C07319=1124.447,364.307,-84.895,-177.079,11.092,149.484
C07320=1124.444,364.554,-84.931,-177.076,11.094,149.483
C07321=1124.440,364.802,-84.967,-177.072,11.097,149.483
C07322=1124.436,365.049,-85.004,-177.069,11.099,149.483
C07323=1124.432,365.296,-85.040,-177.065,11.101,149.483
C07324=1124.429,365.543,-85.076,-177.062,11.104,149.482
C07325=1124.425,365.791,-85.113,-177.059,11.106,149.482
C07326=1124.421,366.038,-85.148,-177.056,11.109,149.482
C07327=1124.417,366.285,-85.185,-177.052,11.111,149.482
C07328=1124.413,366.532,-85.221,-177.050,11.113,149.482
C07329=1124.409,366.779,-85.258,-177.046,11.115,149.481
C07330=1124.406,367.027,-85.294,-177.043,11.118,149.481
C07331=1124.402,367.274,-85.331,-177.039,11.120,149.481
C07332=1124.398,367.522,-85.368,-177.036,11.123,149.480
C07333=1124.394,367.769,-85.403,-177.033,11.125,149.480
C07334=1124.390,368.017,-85.440,-177.029,11.128,149.480
C07335=1124.387,368.264,-85.477,-177.026,11.130,149.480
C07336=1124.383,368.511,-85.513,-177.023,11.132,149.480
C07337=1124.379,368.758,-85.550,-177.020,11.134,149.479
C07338=1124.375,369.005,-85.586,-177.017,11.137,149.479
C07339=1124.372,369.253,-85.623,-177.014,11.139,149.479
C07340=1124.368,369.500,-85.659,-177.010,11.142,149.479
C07341=1124.364,369.747,-85.696,-177.007,11.144,149.479
C07342=1124.360,369.995,-85.733,-177.004,11.146,149.478
C07343=1124.357,370.241,-85.769,-177.001,11.148,149.478
C07344=1124.353,370.489,-85.806,-176.998,11.151,149.478
C07345=1124.349,370.737,-85.843,-176.994,11.153,149.478
C07346=1124.346,370.983,-85.880,-176.991,11.156,149.477
C07347=1124.342,371.231,-85.917,-176.988,11.158,149.477
C07348=1124.338,371.478,-85.953,-176.985,11.160,149.477
C07349=1124.333,371.725,-85.990,-176.982,11.162,149.477
C07350=1124.331,371.973,-86.027,-176.978,11.165,149.477
C07351=1124.327,372.220,-86.064,-176.975,11.167,149.476
C07352=1124.323,372.467,-86.101,-176.972,11.170,149.476
C07353=1124.318,372.714,-86.137,-176.969,11.171,149.476
C07354=1124.315,372.961,-86.174,-176.966,11.174,149.476
C07355=1124.312,373.209,-86.211,-176.963,11.176,149.476
C07356=1124.308,373.456,-86.248,-176.960,11.179,149.476
C07357=1124.303,373.703,-86.285,-176.956,11.182,149.475
C07358=1124.300,373.950,-86.321,-176.954,11.183,149.475
C07359=1124.297,374.198,-86.358,-176.950,11.186,149.475
C07360=1124.292,374.445,-86.395,-176.947,11.188,149.475
C07361=1124.288,374.692,-86.432,-176.944,11.191,149.474
C07362=1124.285,374.939,-86.469,-176.942,11.193,149.474
C07363=1124.282,375.152,-86.501,-176.938,11.195,149.474
C07364=1124.279,375.364,-86.533,-176.936,11.197,149.474
C07365=1124.275,375.577,-86.565,-176.933,11.199,149.474
C07366=1124.272,375.789,-86.597,-176.931,11.201,149.474
C07367=1124.269,376.001,-86.628,-176.928,11.204,149.474
C07368=1124.266,376.214,-86.660,-176.925,11.205,149.473
C07369=1124.262,376.426,-86.691,-176.923,11.207,149.473
C07370=1124.259,376.638,-86.723,-176.921,11.209,149.473
C07371=1124.256,376.886,-86.761,-176.917,11.212,149.473
C07372=1124.252,377.132,-86.798,-176.914,11.214,149.473
C07373=1124.248,377.379,-86.835,-176.911,11.216,149.473
C07374=1124.244,377.626,-86.872,-176.908,11.219,149.473
C07375=1124.241,377.874,-86.910,-176.905,11.221,149.472
C07376=1124.237,378.121,-86.947,-176.902,11.224,149.472
C07377=1124.233,378.368,-86.984,-176.900,11.226,149.472
C07378=1124.229,378.615,-87.021,-176.896,11.228,149.472
C07379=1124.225,378.863,-87.058,-176.893,11.231,149.472
C07380=1124.221,379.110,-87.095,-176.890,11.234,149.472
C07381=1124.218,379.357,-87.133,-176.888,11.236,149.472
C07382=1124.214,379.604,-87.170,-176.884,11.238,149.471
C07383=1124.211,379.852,-87.208,-176.882,11.241,149.471
C07384=1124.207,380.099,-87.245,-176.878,11.243,149.471
C07385=1124.203,380.345,-87.282,-176.876,11.245,149.471
C07386=1124.199,380.593,-87.320,-176.873,11.248,149.471
C07387=1124.196,380.840,-87.357,-176.870,11.251,149.471
C07388=1124.191,381.087,-87.394,-176.867,11.252,149.471
C07389=1124.188,381.334,-87.432,-176.864,11.255,149.471
C07390=1124.184,381.581,-87.469,-176.861,11.258,149.471
C07391=1124.181,381.829,-87.507,-176.858,11.261,149.471
C07392=1124.177,382.076,-87.544,-176.856,11.263,149.471
C07393=1124.174,382.323,-87.582,-176.853,11.265,149.470
C07394=1124.170,382.570,-87.618,-176.850,11.268,149.470
C07395=1124.166,382.817,-87.656,-176.847,11.270,149.470
C07396=1124.163,383.064,-87.694,-176.844,11.273,149.470
C07397=1124.158,383.312,-87.731,-176.841,11.275,149.470
C07398=1124.155,383.559,-87.769,-176.839,11.278,149.470
C07399=1124.151,383.806,-87.807,-176.837,11.280,149.470
C07400=1124.147,384.053,-87.844,-176.836,11.281,149.470
C07401=1124.144,384.300,-87.882,-176.833,11.283,149.470
C07402=1124.140,384.547,-87.919,-176.832,11.285,149.470
C07403=1124.136,384.794,-87.956,-176.830,11.287,149.470
C07404=1124.132,385.041,-87.994,-176.828,11.289,149.471
C07405=1124.129,385.289,-88.033,-176.827,11.291,149.470
C07406=1124.124,385.536,-88.069,-176.825,11.293,149.471
C07407=1124.121,385.783,-88.107,-176.823,11.295,149.471
C07408=1124.117,386.030,-88.145,-176.822,11.297,149.471
C07409=1124.114,386.277,-88.183,-176.820,11.299,149.471
C07410=1124.110,386.524,-88.220,-176.818,11.302,149.471
C07411=1124.106,386.772,-88.258,-176.816,11.304,149.471
C07412=1124.102,387.018,-88.296,-176.815,11.306,149.471
C07413=1124.099,387.265,-88.334,-176.813,11.308,149.471
C07414=1124.095,387.513,-88.371,-176.812,11.311,149.472
C07415=1124.092,387.760,-88.409,-176.810,11.312,149.472
C07416=1124.088,388.007,-88.446,-176.808,11.315,149.472
C07417=1124.084,388.254,-88.485,-176.807,11.317,149.472
C07418=1124.080,388.501,-88.522,-176.805,11.320,149.472
C07419=1124.077,388.713,-88.555,-176.804,11.321,149.472
C07420=1124.074,388.925,-88.587,-176.803,11.323,149.473
C07421=1124.071,389.137,-88.619,-176.801,11.325,149.473
C07422=1124.068,389.349,-88.651,-176.800,11.327,149.473
C07423=1124.065,389.562,-88.684,-176.798,11.330,149.473
C07424=1124.061,389.774,-88.717,-176.797,11.331,149.473
C07425=1124.059,389.987,-88.749,-176.796,11.333,149.474
C07426=1124.054,390.323,-88.801,-176.794,11.337,149.474
C07427=1124.050,390.571,-88.838,-176.792,11.339,149.474
C07428=1124.046,390.817,-88.877,-176.791,11.342,149.474
C07429=1124.042,391.065,-88.915,-176.789,11.344,149.475
C07430=1124.039,391.311,-88.952,-176.788,11.346,149.475
C07431=1124.035,391.559,-88.990,-176.787,11.349,149.475
C07432=1124.031,391.805,-89.028,-176.786,11.352,149.476
C07433=1124.028,392.053,-89.066,-176.784,11.354,149.476
C07434=1124.025,392.300,-89.104,-176.783,11.357,149.476
C07435=1124.020,392.547,-89.142,-176.781,11.360,149.477
C07436=1124.017,392.794,-89.180,-176.780,11.362,149.477
C07437=1124.013,393.041,-89.218,-176.778,11.365,149.477
C07438=1124.010,393.288,-89.256,-176.778,11.367,149.478
C07439=1124.005,393.535,-89.294,-176.776,11.370,149.478
C07440=1124.002,393.782,-89.332,-176.775,11.373,149.478
C07441=1123.998,394.030,-89.370,-176.774,11.376,149.479
C07442=1123.994,394.276,-89.408,-176.772,11.378,149.479
C07443=1123.991,394.524,-89.446,-176.771,11.381,149.480
C07444=1123.987,394.770,-89.484,-176.770,11.384,149.480
C07445=1123.984,395.018,-89.522,-176.768,11.387,149.481
C07446=1123.980,395.265,-89.560,-176.767,11.390,149.481
C07447=1123.976,395.512,-89.598,-176.766,11.393,149.481
C07448=1123.973,395.759,-89.636,-176.765,11.396,149.482
C07449=1123.969,396.005,-89.674,-176.763,11.399,149.482
C07450=1123.965,396.253,-89.713,-176.762,11.402,149.483
C07451=1123.962,396.500,-89.751,-176.761,11.405,149.483
C07452=1123.958,396.747,-89.789,-176.760,11.408,149.484
C07453=1123.954,396.994,-89.827,-176.759,11.411,149.484
C07454=1123.951,397.241,-89.864,-176.758,11.414,149.485
C07455=1123.947,397.488,-89.903,-176.757,11.417,149.485
C07456=1123.943,397.735,-89.941,-176.756,11.420,149.486
C07457=1123.939,397.982,-89.980,-176.755,11.423,149.486
C07458=1123.936,398.229,-90.018,-176.754,11.426,149.487
C07459=1123.932,398.477,-90.056,-176.753,11.429,149.488
C07460=1123.928,398.723,-90.094,-176.751,11.433,149.488
C07461=1123.925,398.970,-90.132,-176.750,11.436,149.489
C07462=1123.922,399.217,-90.171,-176.750,11.439,149.489
C07463=1123.918,399.464,-90.209,-176.749,11.442,149.490
C07464=1123.914,399.712,-90.247,-176.748,11.446,149.491
C07465=1123.911,399.959,-90.285,-176.747,11.449,149.491
C07466=1123.906,400.205,-90.324,-176.746,11.452,149.492
C07467=1123.903,400.452,-90.362,-176.745,11.456,149.493
C07468=1123.899,400.700,-90.400,-176.744,11.460,149.493
C07469=1123.896,400.947,-90.438,-176.743,11.463,149.494
C07470=1123.892,401.193,-90.477,-176.742,11.466,149.494
C07471=1123.889,401.441,-90.515,-176.742,11.469,149.495
C07472=1123.884,401.688,-90.553,-176.741,11.474,149.496
C07473=1123.881,401.934,-90.592,-176.740,11.477,149.497
C07474=1123.877,402.182,-90.631,-176.739,11.480,149.497
C07475=1123.872,402.574,-90.691,-176.738,11.486,149.499
C07476=1123.866,402.967,-90.753,-176.736,11.492,149.500
C07477=1123.860,403.360,-90.813,-176.735,11.498,149.501
C07478=1123.854,403.753,-90.874,-176.734,11.504,149.502
C07479=1123.851,404.000,-90.913,-176.734,11.507,149.503
C07480=1123.847,404.248,-90.952,-176.733,11.512,149.504
C07481=1123.843,404.494,-90.990,-176.732,11.515,149.505
C07482=1123.839,404.741,-91.029,-176.731,11.520,149.506
C07483=1123.836,404.989,-91.067,-176.731,11.523,149.507
C07484=1123.833,405.236,-91.106,-176.731,11.527,149.507
C07485=1123.829,405.482,-91.143,-176.730,11.532,149.508
C07486=1123.825,405.729,-91.183,-176.730,11.535,149.509
C07487=1123.822,405.976,-91.221,-176.729,11.540,149.510
C07488=1123.818,406.223,-91.259,-176.728,11.543,149.511
C07489=1123.814,406.470,-91.298,-176.728,11.548,149.512
C07490=1123.811,406.717,-91.337,-176.727,11.552,149.513
C07491=1123.807,406.965,-91.375,-176.727,11.555,149.514
C07492=1123.804,407.211,-91.414,-176.727,11.560,149.515
C07493=1123.800,407.458,-91.452,-176.726,11.564,149.516
C07494=1123.796,407.705,-91.491,-176.726,11.569,149.517
C07495=1123.793,407.952,-91.529,-176.725,11.573,149.518
C07496=1123.789,408.199,-91.568,-176.725,11.577,149.519
C07497=1123.785,408.446,-91.607,-176.724,11.582,149.520
C07498=1123.782,408.693,-91.645,-176.724,11.586,149.521
C07499=1123.778,408.940,-91.684,-176.724,11.591,149.522
C07500=1123.775,409.187,-91.722,-176.724,11.595,149.523
C07501=1123.771,409.434,-91.762,-176.723,11.599,149.524
C07502=1123.767,409.681,-91.800,-176.723,11.604,149.526
C07503=1123.764,409.927,-91.839,-176.723,11.608,149.527
C07504=1123.760,410.175,-91.877,-176.722,11.613,149.528
C07505=1123.756,410.422,-91.916,-176.722,11.618,149.529
C07506=1123.753,410.669,-91.956,-176.722,11.622,149.530
C07507=1123.749,410.916,-91.993,-176.722,11.627,149.531
C07508=1123.745,411.163,-92.032,-176.721,11.632,149.532
C07509=1123.742,411.409,-92.072,-176.721,11.637,149.534
C07510=1123.739,411.657,-92.110,-176.721,11.641,149.535
C07511=1123.735,411.904,-92.149,-176.721,11.646,149.536
C07512=1123.731,412.150,-92.188,-176.720,11.651,149.537
C07513=1123.728,412.397,-92.226,-176.720,11.656,149.538
C07514=1123.724,412.644,-92.265,-176.721,11.660,149.540
C07515=1123.720,412.891,-92.304,-176.721,11.665,149.541
C07516=1123.717,413.138,-92.343,-176.720,11.670,149.542
C07517=1123.714,413.385,-92.381,-176.720,11.675,149.544
C07518=1123.710,413.632,-92.421,-176.720,11.681,149.545
C07519=1123.706,413.879,-92.460,-176.720,11.686,149.546
C07520=1123.703,414.126,-92.499,-176.721,11.690,149.548
C07521=1123.701,414.373,-92.537,-176.721,11.696,149.549
C07522=1123.699,414.620,-92.576,-176.721,11.701,149.550
C07523=1123.697,414.867,-92.614,-176.721,11.706,149.552
C07524=1123.696,415.114,-92.652,-176.721,11.712,149.553
C07525=1123.696,415.361,-92.691,-176.721,11.717,149.554
C07526=1123.696,415.608,-92.730,-176.721,11.722,149.556
C07527=1123.697,415.820,-92.763,-176.722,11.727,149.557
C07528=1123.698,416.032,-92.795,-176.722,11.731,149.558
C07529=1123.700,416.243,-92.828,-176.722,11.736,149.560
C07530=1123.702,416.455,-92.861,-176.722,11.740,149.561
C07531=1123.704,416.667,-92.893,-176.722,11.746,149.562
C07532=1123.707,416.879,-92.926,-176.723,11.750,149.564
C07533=1123.710,417.091,-92.959,-176.723,11.754,149.565
C07534=1123.714,417.303,-92.991,-176.723,11.760,149.566
C07535=1123.295,417.302,-93.053,-176.716,11.764,149.566
C07536=1123.291,417.091,-93.022,-176.716,11.759,149.564
C07537=1123.288,416.879,-92.988,-176.715,11.754,149.563
C07538=1123.285,416.667,-92.956,-176.715,11.750,149.562
C07539=1123.283,416.455,-92.923,-176.715,11.745,149.560
C07540=1123.281,416.243,-92.890,-176.715,11.741,149.559
C07541=1123.279,416.032,-92.858,-176.715,11.735,149.558
C07542=1123.278,415.819,-92.825,-176.715,11.731,149.557
C07543=1123.277,415.608,-92.792,-176.714,11.727,149.555
C07544=1123.277,415.361,-92.754,-176.714,11.721,149.554
C07545=1123.277,415.114,-92.715,-176.714,11.716,149.552
C07546=1123.279,414.867,-92.677,-176.713,11.711,149.551
C07547=1123.279,414.620,-92.637,-176.714,11.705,149.550
C07548=1123.281,414.373,-92.599,-176.713,11.700,149.548
C07549=1123.284,414.126,-92.560,-176.714,11.695,149.547
C07550=1123.286,413.879,-92.522,-176.714,11.690,149.546
C07551=1123.290,413.632,-92.483,-176.714,11.684,149.544
C07552=1123.294,413.385,-92.444,-176.714,11.679,149.543
C07553=1123.297,413.138,-92.405,-176.714,11.674,149.542
C07554=1123.301,412.891,-92.366,-176.714,11.669,149.540
C07555=1123.305,412.644,-92.328,-176.714,11.664,149.539
C07556=1123.309,412.397,-92.288,-176.715,11.659,149.538
C07557=1123.312,412.151,-92.250,-176.714,11.655,149.537
C07558=1123.315,411.904,-92.211,-176.715,11.650,149.535
C07559=1123.319,411.656,-92.172,-176.715,11.645,149.534
C07560=1123.323,411.409,-92.133,-176.715,11.640,149.533
C07561=1123.326,411.163,-92.094,-176.716,11.635,149.532
C07562=1123.330,410.916,-92.056,-176.715,11.631,149.531
C07563=1123.334,410.669,-92.017,-176.716,11.626,149.529
C07564=1123.337,410.422,-91.978,-176.716,11.621,149.528
C07565=1123.341,410.174,-91.939,-176.716,11.616,149.527
C07566=1123.344,409.927,-91.900,-176.716,11.612,149.526
C07567=1123.348,409.681,-91.862,-176.717,11.607,149.525
C07568=1123.352,409.434,-91.823,-176.718,11.602,149.524
C07569=1123.355,409.187,-91.784,-176.717,11.598,149.523
C07570=1123.358,408.940,-91.746,-176.718,11.594,149.522
C07571=1123.362,408.693,-91.707,-176.719,11.589,149.521
C07572=1123.366,408.446,-91.668,-176.719,11.585,149.520
C07573=1123.369,408.199,-91.630,-176.719,11.580,149.519
C07574=1123.373,407.952,-91.591,-176.720,11.576,149.517
C07575=1123.377,407.705,-91.552,-176.720,11.572,149.517
C07576=1123.380,407.459,-91.514,-176.721,11.567,149.515
C07577=1123.384,407.211,-91.476,-176.721,11.564,149.515
C07578=1123.388,406.964,-91.436,-176.722,11.559,149.513
C07579=1123.391,406.717,-91.398,-176.723,11.554,149.513
C07580=1123.395,406.470,-91.359,-176.723,11.551,149.512
C07581=1123.399,406.223,-91.322,-176.724,11.546,149.511
C07582=1123.402,405.976,-91.282,-176.724,11.542,149.510
C07583=1123.406,405.729,-91.244,-176.725,11.538,149.509
C07584=1123.409,405.482,-91.205,-176.725,11.534,149.508
C07585=1123.414,405.235,-91.167,-176.726,11.530,149.507
C07586=1123.416,404.989,-91.128,-176.726,11.526,149.506
C07587=1123.420,404.741,-91.090,-176.727,11.523,149.505
C07588=1123.423,404.494,-91.051,-176.728,11.518,149.504
C07589=1123.428,404.247,-91.013,-176.728,11.515,149.504
C07590=1123.431,404.001,-90.974,-176.729,11.510,149.503
C07591=1123.435,403.753,-90.936,-176.730,11.507,149.502
C07592=1123.438,403.542,-90.902,-176.731,11.503,149.501
C07593=1123.441,403.329,-90.870,-176.731,11.500,149.501
C07594=1123.444,403.117,-90.836,-176.732,11.497,149.500
C07595=1123.448,402.905,-90.804,-176.733,11.493,149.499
C07596=1123.450,402.694,-90.771,-176.734,11.490,149.499
C07597=1123.453,402.481,-90.738,-176.734,11.488,149.498
C07598=1123.456,402.269,-90.705,-176.735,11.485,149.497
C07599=1123.459,402.057,-90.672,-176.735,11.481,149.497
C07600=1123.463,401.810,-90.633,-176.736,11.478,149.496
C07601=1123.467,401.563,-90.596,-176.737,11.474,149.495
C07602=1123.471,401.316,-90.556,-176.738,11.470,149.495
C07603=1123.474,401.069,-90.518,-176.739,11.467,149.494
C07604=1123.479,400.822,-90.480,-176.740,11.464,149.493
C07605=1123.481,400.575,-90.442,-176.741,11.460,149.492
C07606=1123.485,400.328,-90.403,-176.742,11.456,149.492
C07607=1123.489,400.081,-90.365,-176.743,11.453,149.491
C07608=1123.493,399.834,-90.327,-176.743,11.450,149.491
C07609=1123.496,399.587,-90.288,-176.745,11.446,149.490
C07610=1123.500,399.340,-90.251,-176.746,11.443,149.489
C07611=1123.504,399.093,-90.212,-176.747,11.440,149.489
C07612=1123.507,398.846,-90.174,-176.748,11.436,149.488
C07613=1123.511,398.599,-90.135,-176.749,11.433,149.488
C07614=1123.514,398.352,-90.097,-176.749,11.430,149.487
C07615=1123.518,398.104,-90.059,-176.751,11.426,149.486
C07616=1123.522,397.858,-90.021,-176.752,11.423,149.486
C07617=1123.526,397.610,-89.983,-176.753,11.420,149.485
C07618=1123.529,397.364,-89.944,-176.754,11.417,149.485
C07619=1123.533,397.117,-89.906,-176.755,11.414,149.484
C07620=1123.536,396.869,-89.868,-176.757,11.411,149.484
C07621=1123.540,396.623,-89.830,-176.758,11.408,149.483
C07622=1123.544,396.375,-89.792,-176.759,11.405,149.483
C07623=1123.547,396.128,-89.754,-176.760,11.402,149.482
C07624=1123.551,395.881,-89.716,-176.761,11.399,149.482
C07625=1123.555,395.634,-89.678,-176.762,11.396,149.481
C07626=1123.559,395.388,-89.640,-176.764,11.393,149.481
C07627=1123.562,395.140,-89.601,-176.765,11.390,149.480
C07628=1123.566,394.893,-89.563,-176.767,11.387,149.480
C07629=1123.569,394.647,-89.525,-176.768,11.384,149.480
C07630=1123.573,394.399,-89.487,-176.769,11.381,149.479
C07631=1123.577,394.152,-89.449,-176.770,11.378,149.479
C07632=1123.580,393.905,-89.411,-176.771,11.376,149.478
C07633=1123.584,393.658,-89.373,-176.772,11.373,149.478
C07634=1123.588,393.411,-89.335,-176.774,11.371,149.478
C07635=1123.591,393.164,-89.297,-176.775,11.368,149.477
C07636=1123.596,392.917,-89.259,-176.777,11.365,149.477
C07637=1123.599,392.670,-89.221,-176.778,11.363,149.477
C07638=1123.603,392.423,-89.184,-176.780,11.360,149.476
C07639=1123.607,392.175,-89.145,-176.781,11.357,149.476
C07640=1123.610,391.928,-89.107,-176.782,11.354,149.476
C07641=1123.614,391.682,-89.070,-176.784,11.352,149.475
C07642=1123.617,391.434,-89.032,-176.786,11.349,149.475
C07643=1123.621,391.187,-88.994,-176.787,11.346,149.475
C07644=1123.625,390.940,-88.956,-176.789,11.344,149.474
C07645=1123.628,390.694,-88.918,-176.789,11.342,149.474
C07646=1123.632,390.446,-88.879,-176.791,11.339,149.474
C07647=1123.636,390.199,-88.842,-176.793,11.337,149.474
C07648=1123.640,389.922,-88.799,-176.794,11.334,149.473
C07649=1123.644,389.644,-88.757,-176.796,11.331,149.473
C07650=1123.648,389.367,-88.714,-176.798,11.328,149.473
C07651=1123.652,389.089,-88.672,-176.800,11.326,149.473
C07652=1123.656,388.842,-88.634,-176.802,11.323,149.472
C07653=1123.660,388.594,-88.597,-176.803,11.322,149.472
C07654=1123.663,388.348,-88.559,-176.804,11.319,149.472
C07655=1123.667,388.101,-88.521,-176.806,11.317,149.472
C07656=1123.671,387.854,-88.483,-176.808,11.314,149.472
C07657=1123.674,387.606,-88.445,-176.809,11.312,149.471
C07658=1123.678,387.360,-88.408,-176.811,11.310,149.471
C07659=1123.682,387.112,-88.370,-176.813,11.308,149.471
C07660=1123.685,386.865,-88.333,-176.815,11.305,149.471
C07661=1123.689,386.618,-88.295,-176.816,11.304,149.471
C07662=1123.693,386.371,-88.257,-176.818,11.301,149.471
C07663=1123.697,386.123,-88.219,-176.820,11.299,149.471
C07664=1123.700,385.877,-88.182,-176.821,11.297,149.471
C07665=1123.704,385.630,-88.144,-176.823,11.295,149.470
C07666=1123.707,385.383,-88.106,-176.825,11.293,149.470
C07667=1123.711,385.135,-88.069,-176.827,11.291,149.470
C07668=1123.715,384.888,-88.031,-176.828,11.289,149.470
C07669=1123.719,384.641,-87.993,-176.830,11.287,149.470
C07670=1123.723,384.394,-87.956,-176.832,11.284,149.470
C07671=1123.726,384.147,-87.918,-176.834,11.282,149.470
C07672=1123.730,383.900,-87.881,-176.835,11.281,149.470
C07673=1123.734,383.653,-87.844,-176.838,11.279,149.470
C07674=1123.737,383.405,-87.806,-176.839,11.276,149.470
C07675=1123.741,383.159,-87.768,-176.842,11.274,149.470
C07676=1123.745,382.911,-87.731,-176.845,11.272,149.470
C07677=1123.749,382.664,-87.693,-176.848,11.269,149.470
C07678=1123.752,382.417,-87.655,-176.851,11.266,149.470
C07679=1123.756,382.170,-87.618,-176.854,11.265,149.470
C07680=1123.760,381.923,-87.581,-176.856,11.262,149.470
C07681=1123.763,381.675,-87.543,-176.859,11.259,149.470
C07682=1123.767,381.429,-87.506,-176.862,11.257,149.471
C07683=1123.771,381.181,-87.469,-176.865,11.254,149.471
C07684=1123.774,380.934,-87.431,-176.868,11.252,149.471
C07685=1123.778,380.686,-87.394,-176.871,11.249,149.471
C07686=1123.782,380.440,-87.356,-176.873,11.247,149.471
C07687=1123.786,380.193,-87.319,-176.877,11.245,149.471
C07688=1123.789,379.945,-87.281,-176.880,11.242,149.471
C07689=1123.793,379.698,-87.245,-176.883,11.239,149.471
C07690=1123.797,379.452,-87.207,-176.885,11.237,149.471
C07691=1123.800,379.204,-87.170,-176.888,11.235,149.472
C07692=1123.807,378.810,-87.111,-176.893,11.231,149.472
C07693=1123.812,378.416,-87.051,-176.898,11.227,149.472
C07694=1123.819,378.021,-86.991,-176.903,11.223,149.472
C07695=1123.824,377.627,-86.932,-176.907,11.219,149.472
C07696=1123.828,377.380,-86.895,-176.911,11.217,149.473
C07697=1123.832,377.133,-86.858,-176.913,11.215,149.473
C07698=1123.836,376.885,-86.821,-176.916,11.212,149.473
C07699=1123.839,376.639,-86.784,-176.920,11.210,149.473
C07700=1123.843,376.426,-86.752,-176.922,11.208,149.473
C07701=1123.846,376.215,-86.720,-176.924,11.206,149.473
C07702=1123.850,376.002,-86.688,-176.927,11.203,149.473
C07703=1123.853,375.790,-86.656,-176.930,11.202,149.474
C07704=1123.856,375.577,-86.625,-176.932,11.200,149.474
C07705=1123.858,375.365,-86.593,-176.935,11.198,149.474
C07706=1123.862,375.152,-86.561,-176.938,11.195,149.474
C07707=1123.865,374.941,-86.529,-176.941,11.193,149.474
C07708=1123.869,374.693,-86.492,-176.944,11.191,149.474
C07709=1123.873,374.445,-86.455,-176.947,11.189,149.475
C07710=1123.877,374.198,-86.419,-176.949,11.186,149.475
C07711=1123.880,373.951,-86.381,-176.953,11.184,149.475
C07712=1123.884,373.704,-86.344,-176.956,11.181,149.475
C07713=1123.888,373.457,-86.307,-176.959,11.179,149.475
C07714=1123.892,373.210,-86.271,-176.962,11.177,149.476
C07715=1123.896,372.963,-86.234,-176.965,11.175,149.476
C07716=1123.899,372.715,-86.197,-176.969,11.172,149.476
C07717=1123.903,372.468,-86.160,-176.972,11.170,149.476
C07718=1123.907,372.221,-86.123,-176.975,11.167,149.476
C07719=1123.910,371.974,-86.087,-176.977,11.165,149.476
C07720=1123.914,371.726,-86.050,-176.981,11.163,149.477
C07721=1123.918,371.479,-86.013,-176.984,11.160,149.477
C07722=1123.922,371.231,-85.976,-176.987,11.158,149.477
C07723=1123.925,370.985,-85.940,-176.991,11.155,149.477
C07724=1123.929,370.737,-85.903,-176.993,11.154,149.478
C07725=1123.933,370.489,-85.866,-176.997,11.151,149.478
C07726=1123.936,370.243,-85.830,-177.000,11.149,149.478
C07727=1123.940,369.995,-85.793,-177.003,11.146,149.478
C07728=1123.944,369.748,-85.756,-177.007,11.144,149.478
C07729=1123.948,369.501,-85.720,-177.010,11.141,149.479
C07730=1123.952,369.254,-85.683,-177.012,11.140,149.479
C07731=1123.956,369.006,-85.646,-177.016,11.137,149.479
C07732=1123.959,368.759,-85.610,-177.019,11.135,149.479
C07733=1123.963,368.512,-85.573,-177.023,11.132,149.480
C07734=1123.967,368.264,-85.536,-177.026,11.130,149.480
C07735=1123.971,368.017,-85.501,-177.029,11.128,149.480
C07736=1123.975,367.770,-85.464,-177.033,11.125,149.480
C07737=1123.978,367.523,-85.428,-177.036,11.123,149.480
C07738=1123.982,367.276,-85.391,-177.039,11.121,149.481
C07739=1123.986,367.027,-85.355,-177.042,11.118,149.481
C07740=1123.990,366.780,-85.318,-177.045,11.116,149.481
C07741=1123.994,366.533,-85.281,-177.049,11.113,149.481
C07742=1123.997,366.286,-85.245,-177.052,11.111,149.482
C07743=1124.001,366.038,-85.209,-177.056,11.109,149.482
C07744=1124.005,365.791,-85.172,-177.059,11.106,149.482
C07745=1124.009,365.544,-85.136,-177.062,11.104,149.482
C07746=1124.013,365.297,-85.100,-177.065,11.101,149.483
C07747=1124.017,365.050,-85.063,-177.068,11.100,149.483
C07748=1124.020,364.802,-85.028,-177.071,11.097,149.483
C07749=1124.024,364.555,-84.991,-177.075,11.095,149.483
C07750=1124.028,364.308,-84.954,-177.078,11.093,149.484
C07751=1124.032,364.060,-84.918,-177.082,11.090,149.484
C07752=1124.035,363.813,-84.882,-177.085,11.088,149.484
C07753=1124.039,363.565,-84.846,-177.088,11.085,149.484
C07754=1124.043,363.318,-84.809,-177.092,11.083,149.485
C07755=1124.046,363.070,-84.774,-177.095,11.081,149.485
C07756=1124.050,362.858,-84.743,-177.098,11.079,149.485
C07757=1124.053,362.646,-84.712,-177.101,11.076,149.485
C07758=1124.056,362.433,-84.680,-177.104,11.074,149.485
C07759=1124.060,362.221,-84.649,-177.107,11.072,149.486
C07760=1124.063,362.009,-84.618,-177.110,11.070,149.486
C07761=1124.067,361.796,-84.588,-177.112,11.069,149.486
C07762=1124.070,361.583,-84.557,-177.116,11.066,149.486
C07763=1124.073,361.371,-84.525,-177.118,11.064,149.487
C07764=1124.076,361.124,-84.489,-177.122,11.062,149.487
C07765=1124.080,360.876,-84.454,-177.125,11.059,149.487
C07766=1124.084,360.629,-84.417,-177.129,11.057,149.488
C07767=1124.088,360.382,-84.381,-177.132,11.055,149.488
C07768=1124.091,360.134,-84.346,-177.135,11.052,149.488
C07769=1124.096,359.887,-84.310,-177.138,11.050,149.488
C07770=1124.100,359.640,-84.274,-177.142,11.048,149.489
C07771=1124.103,359.393,-84.238,-177.145,11.045,149.489
C07772=1124.107,359.145,-84.202,-177.149,11.043,149.489
C07773=1124.111,358.897,-84.166,-177.153,11.040,149.489
C07774=1124.115,358.650,-84.130,-177.156,11.037,149.489
C07775=1124.118,358.403,-84.095,-177.160,11.035,149.490
C07776=1124.122,358.155,-84.059,-177.163,11.033,149.490
C07777=1124.126,357.908,-84.023,-177.166,11.030,149.490
C07778=1124.130,357.660,-83.987,-177.170,11.028,149.490
C07779=1124.134,357.413,-83.952,-177.173,11.025,149.491
C07780=1124.137,357.166,-83.915,-177.177,11.023,149.491
C07781=1124.142,356.918,-83.879,-177.180,11.021,149.491
C07782=1124.146,356.671,-83.844,-177.183,11.018,149.492
C07783=1124.149,356.424,-83.809,-177.187,11.016,149.492
C07784=1124.153,356.176,-83.773,-177.190,11.013,149.492
C07785=1124.157,355.929,-83.737,-177.194,11.010,149.492
C07786=1124.160,355.681,-83.702,-177.198,11.008,149.493
C07787=1124.164,355.434,-83.666,-177.201,11.006,149.493
C07788=1124.168,355.186,-83.630,-177.205,11.003,149.493
C07789=1124.173,354.939,-83.595,-177.208,11.001,149.493
C07790=1124.176,354.692,-83.560,-177.211,10.998,149.494
C07791=1124.180,354.444,-83.524,-177.215,10.996,149.494
C07792=1124.184,354.197,-83.488,-177.219,10.993,149.494
C07793=1124.187,353.949,-83.453,-177.222,10.990,149.494
C07794=1124.191,353.702,-83.417,-177.225,10.988,149.495
C07795=1124.195,353.455,-83.382,-177.229,10.985,149.495
C07796=1124.199,353.207,-83.347,-177.232,10.983,149.495
C07797=1124.203,352.960,-83.311,-177.236,10.980,149.495
C07798=1124.207,352.712,-83.276,-177.240,10.978,149.496
C07799=1124.211,352.464,-83.240,-177.243,10.975,149.496
C07800=1124.215,352.217,-83.205,-177.246,10.973,149.496
C07801=1124.219,351.970,-83.169,-177.250,10.971,149.497
C07802=1124.223,351.722,-83.134,-177.254,10.967,149.497
C07803=1124.226,351.475,-83.098,-177.257,10.965,149.497
C07804=1124.231,351.227,-83.064,-177.261,10.962,149.497
C07805=1124.235,350.980,-83.028,-177.264,10.960,149.497
C07806=1124.237,350.732,-82.993,-177.268,10.957,149.498
C07807=1124.241,350.485,-82.958,-177.272,10.955,149.498
C07808=1124.246,350.237,-82.923,-177.275,10.952,149.498
C07809=1124.249,349.990,-82.888,-177.279,10.949,149.498
C07810=1124.253,349.742,-82.852,-177.282,10.946,149.499
C07811=1124.258,349.495,-82.818,-177.285,10.944,149.499
C07812=1124.261,349.282,-82.787,-177.289,10.941,149.499
C07813=1124.264,349.070,-82.757,-177.291,10.940,149.499
C07814=1124.267,348.857,-82.726,-177.294,10.938,149.499
C07815=1124.270,348.645,-82.697,-177.297,10.935,149.500
C07816=1124.274,348.432,-82.666,-177.299,10.933,149.500
C07817=1124.277,348.219,-82.637,-177.303,10.931,149.500
C07818=1124.281,348.007,-82.606,-177.305,10.929,149.500
C07819=1124.284,347.794,-82.577,-177.308,10.927,149.500
C07820=1124.288,347.547,-82.541,-177.311,10.925,149.501
C07821=1124.292,347.299,-82.506,-177.314,10.922,149.501
C07822=1124.296,347.052,-82.471,-177.318,10.920,149.501
C07823=1124.300,346.804,-82.436,-177.321,10.917,149.501
C07824=1124.304,346.556,-82.401,-177.324,10.915,149.502
C07825=1124.308,346.309,-82.366,-177.327,10.912,149.502
C07826=1124.311,346.062,-82.331,-177.330,10.910,149.502
C07827=1124.316,345.814,-82.297,-177.334,10.907,149.502
C07828=1124.320,345.566,-82.262,-177.337,10.905,149.502
C07829=1124.323,345.319,-82.227,-177.340,10.902,149.502
C07830=1124.327,345.071,-82.193,-177.344,10.900,149.503
C07831=1124.331,344.824,-82.157,-177.347,10.897,149.503
C07832=1124.335,344.576,-82.122,-177.350,10.895,149.503
C07833=1124.339,344.328,-82.088,-177.353,10.892,149.503
C07834=1124.343,344.081,-82.052,-177.356,10.890,149.503
C07835=1124.347,343.834,-82.018,-177.359,10.888,149.504
C07836=1124.351,343.586,-81.984,-177.363,10.886,149.504
C07837=1124.355,343.339,-81.948,-177.365,10.883,149.504
C07838=1124.358,343.091,-81.914,-177.369,10.880,149.504
C07839=1124.363,342.844,-81.880,-177.372,10.878,149.504
C07840=1124.367,342.596,-81.845,-177.375,10.875,149.505
C07841=1124.370,342.348,-81.810,-177.379,10.873,149.505
C07842=1124.374,342.101,-81.775,-177.382,10.870,149.505
C07843=1124.378,341.853,-81.741,-177.385,10.868,149.505
C07844=1124.382,341.606,-81.707,-177.388,10.865,149.505
C07845=1124.386,341.358,-81.672,-177.392,10.863,149.506
C07846=1124.390,341.111,-81.637,-177.395,10.860,149.506
C07847=1124.394,340.863,-81.602,-177.398,10.858,149.506
C07848=1124.398,340.616,-81.568,-177.401,10.855,149.506
C07849=1124.402,340.367,-81.533,-177.404,10.853,149.506
C07850=1124.406,340.120,-81.499,-177.408,10.850,149.507
C07851=1124.410,339.872,-81.464,-177.411,10.848,149.507
C07852=1124.414,339.625,-81.431,-177.414,10.845,149.507
C07853=1124.418,339.377,-81.396,-177.417,10.842,149.507
C07854=1124.422,339.130,-81.361,-177.420,10.841,149.507
C07855=1124.426,338.882,-81.327,-177.423,10.838,149.508
C07856=1124.430,338.634,-81.293,-177.427,10.836,149.508
C07857=1124.434,338.387,-81.259,-177.430,10.833,149.508
C07858=1124.438,338.139,-81.224,-177.433,10.831,149.508
C07859=1124.442,337.892,-81.190,-177.436,10.828,149.508
C07860=1124.446,337.644,-81.155,-177.439,10.826,149.509
C07861=1124.450,337.397,-81.121,-177.443,10.823,149.509
C07862=1124.454,337.149,-81.086,-177.446,10.820,149.509
C07863=1124.457,336.902,-81.053,-177.449,10.818,149.509
C07864=1124.461,336.653,-81.018,-177.452,10.816,149.509
C07865=1124.465,336.406,-80.984,-177.456,10.813,149.510
C07866=1124.470,336.159,-80.949,-177.459,10.810,149.510
C07867=1124.473,335.911,-80.915,-177.462,10.808,149.510
C07868=1124.476,335.698,-80.886,-177.465,10.806,149.510
C07869=1124.480,335.486,-80.857,-177.467,10.804,149.510
C07870=1124.483,335.273,-80.828,-177.470,10.802,149.511
C07871=1124.487,335.060,-80.798,-177.472,10.800,149.511
C07872=1124.490,334.847,-80.768,-177.476,10.797,149.511
C07873=1124.494,334.634,-80.739,-177.478,10.795,149.511
C07874=1124.497,334.422,-80.710,-177.481,10.794,149.511
C07875=1124.500,334.209,-80.681,-177.484,10.791,149.511
C07876=1124.504,333.962,-80.647,-177.487,10.788,149.512
C07877=1124.508,333.714,-80.612,-177.490,10.786,149.512
C07878=1124.512,333.466,-80.579,-177.493,10.783,149.512
C07879=1124.516,333.219,-80.545,-177.497,10.781,149.512
C07880=1124.520,332.971,-80.510,-177.500,10.778,149.512
C07881=1124.524,332.723,-80.477,-177.503,10.777,149.513
C07882=1124.528,332.476,-80.443,-177.505,10.774,149.513
C07883=1124.532,332.228,-80.409,-177.509,10.771,149.513
C07884=1124.536,331.980,-80.375,-177.512,10.769,149.513
C07885=1124.540,331.733,-80.342,-177.515,10.766,149.513
C07886=1124.544,331.484,-80.307,-177.518,10.764,149.513
C07887=1124.548,331.237,-80.274,-177.522,10.761,149.514
C07888=1124.552,330.990,-80.240,-177.525,10.759,149.514
C07889=1124.555,330.741,-80.206,-177.528,10.756,149.514
C07890=1124.560,330.494,-80.172,-177.531,10.754,149.514
C07891=1124.564,330.246,-80.139,-177.535,10.751,149.514
C07892=1124.568,329.999,-80.105,-177.538,10.749,149.515
C07893=1124.572,329.751,-80.071,-177.541,10.746,149.515
C07894=1124.575,329.504,-80.037,-177.544,10.743,149.515
C07895=1124.580,329.256,-80.004,-177.547,10.741,149.515
C07896=1124.583,329.008,-79.969,-177.550,10.738,149.515
C07897=1124.588,328.760,-79.936,-177.554,10.736,149.516
C07898=1124.591,328.513,-79.902,-177.556,10.734,149.516
C07899=1124.596,328.265,-79.869,-177.560,10.732,149.516
C07900=1124.600,328.017,-79.835,-177.563,10.729,149.516
C07901=1124.604,327.769,-79.801,-177.566,10.726,149.516
C07902=1124.608,327.522,-79.768,-177.569,10.724,149.517
C07903=1124.612,327.275,-79.734,-177.572,10.721,149.517
C07904=1124.616,327.027,-79.701,-177.576,10.719,149.517
C07905=1124.619,326.778,-79.667,-177.579,10.716,149.517
C07906=1124.623,326.531,-79.634,-177.582,10.714,149.517
C07907=1124.627,326.284,-79.600,-177.585,10.711,149.517
C07908=1124.632,326.036,-79.567,-177.588,10.709,149.518
C07909=1124.636,325.788,-79.533,-177.592,10.706,149.518
C07910=1124.640,325.540,-79.499,-177.595,10.703,149.518
C07911=1124.644,325.292,-79.466,-177.598,10.701,149.518
C07912=1124.648,325.045,-79.433,-177.601,10.699,149.519
C07913=1124.652,324.797,-79.400,-177.604,10.696,149.519
C07914=1124.656,324.550,-79.366,-177.607,10.694,149.519
C07915=1124.660,324.302,-79.333,-177.610,10.692,149.519
C07916=1124.663,324.054,-79.299,-177.613,10.689,149.519
C07917=1124.668,323.806,-79.266,-177.617,10.686,149.519
C07918=1124.672,323.558,-79.233,-177.620,10.684,149.520
C07919=1124.676,323.310,-79.200,-177.623,10.681,149.520
C07920=1124.680,323.063,-79.166,-177.626,10.679,149.520
C07921=1124.684,322.816,-79.133,-177.629,10.676,149.520
C07922=1124.687,322.567,-79.099,-177.632,10.674,149.520
C07923=1124.692,322.319,-79.066,-177.636,10.671,149.521
C07924=1124.694,322.107,-79.038,-177.638,10.669,149.521
C07925=1124.698,321.893,-79.010,-177.641,10.667,149.521
C07926=1124.702,321.681,-78.981,-177.644,10.665,149.521
C07927=1124.706,321.468,-78.952,-177.646,10.663,149.521
C07928=1124.709,321.256,-78.924,-177.649,10.660,149.521
C07929=1124.712,321.042,-78.896,-177.651,10.658,149.521
C07930=1124.716,320.829,-78.867,-177.655,10.656,149.522
C07931=1124.719,320.617,-78.839,-177.657,10.654,149.522
C07932=1124.723,320.369,-78.805,-177.660,10.651,149.522
C07933=1124.727,320.121,-78.772,-177.663,10.649,149.522
C07934=1124.731,319.874,-78.739,-177.667,10.646,149.522
C07935=1124.736,319.625,-78.707,-177.670,10.644,149.523
C07936=1124.740,319.377,-78.674,-177.673,10.641,149.523
C07937=1124.743,319.130,-78.641,-177.676,10.638,149.523
C07938=1124.747,318.882,-78.608,-177.680,10.636,149.523
C07939=1124.751,318.634,-78.574,-177.682,10.634,149.523
C07940=1124.755,318.386,-78.541,-177.685,10.632,149.524
C07941=1124.759,318.138,-78.508,-177.689,10.629,149.524
C07942=1124.762,317.891,-78.475,-177.691,10.626,149.524
C07943=1124.767,317.643,-78.443,-177.695,10.624,149.524
C07944=1124.771,317.395,-78.410,-177.698,10.621,149.524
C07945=1124.775,317.147,-78.377,-177.701,10.619,149.524
C07946=1124.779,316.900,-78.344,-177.704,10.616,149.525
C07947=1124.783,316.651,-78.312,-177.707,10.613,149.525
C07948=1124.787,316.404,-78.278,-177.711,10.611,149.525
C07949=1124.791,316.156,-78.245,-177.714,10.608,149.525
C07950=1124.795,315.909,-78.213,-177.717,10.606,149.525
C07951=1124.799,315.660,-78.180,-177.720,10.603,149.526
C07952=1124.803,315.412,-78.147,-177.723,10.601,149.526
C07953=1124.807,315.165,-78.114,-177.726,10.598,149.526
C07954=1124.812,314.917,-78.083,-177.729,10.597,149.526
C07955=1124.816,314.670,-78.049,-177.732,10.594,149.526
C07956=1124.820,314.422,-78.016,-177.735,10.591,149.527
C07957=1124.824,314.174,-77.984,-177.738,10.589,149.527
C07958=1124.828,313.926,-77.951,-177.742,10.586,149.527
C07959=1124.832,313.678,-77.919,-177.745,10.584,149.527
C07960=1124.836,313.430,-77.886,-177.748,10.581,149.527
C07961=1124.840,313.182,-77.854,-177.751,10.578,149.527
C07962=1124.844,312.935,-77.821,-177.754,10.576,149.527
C07963=1124.848,312.687,-77.788,-177.757,10.573,149.528
C07964=1124.852,312.439,-77.756,-177.760,10.570,149.528
C07965=1124.856,312.191,-77.723,-177.764,10.568,149.528
C07966=1124.860,311.943,-77.691,-177.767,10.566,149.528
C07967=1124.864,311.695,-77.659,-177.770,10.563,149.528
C07968=1124.868,311.448,-77.626,-177.773,10.561,149.529
C07969=1124.872,311.200,-77.594,-177.776,10.558,149.529
C07970=1124.876,310.952,-77.561,-177.779,10.556,149.529
C07971=1124.881,310.704,-77.529,-177.782,10.554,149.529
C07972=1124.884,310.456,-77.496,-177.785,10.551,149.529
C07973=1124.889,310.208,-77.464,-177.789,10.548,149.530
C07974=1124.893,309.961,-77.432,-177.791,10.546,149.530
C07975=1124.897,309.713,-77.399,-177.795,10.543,149.530
C07976=1124.901,309.465,-77.367,-177.798,10.540,149.530
C07977=1124.905,309.216,-77.335,-177.801,10.538,149.530
C07978=1124.909,308.969,-77.302,-177.804,10.535,149.531
C07979=1124.913,308.721,-77.270,-177.807,10.533,149.531
C07980=1124.917,308.508,-77.242,-177.810,10.531,149.531
C07981=1124.920,308.295,-77.215,-177.812,10.529,149.531
C07982=1124.924,308.081,-77.187,-177.815,10.526,149.531
C07983=1124.927,307.869,-77.159,-177.818,10.524,149.531
C07984=1124.930,307.656,-77.132,-177.821,10.522,149.531
C07985=1124.934,307.442,-77.104,-177.823,10.520,149.532
C07986=1124.938,307.230,-77.077,-177.825,10.518,149.532
C07987=1124.941,307.017,-77.049,-177.829,10.515,149.532
C07988=1124.945,306.768,-77.017,-177.832,10.513,149.532
C07989=1124.949,306.521,-76.984,-177.834,10.511,149.532
C07990=1124.953,306.273,-76.952,-177.837,10.508,149.532
C07991=1124.958,306.025,-76.920,-177.841,10.506,149.533
C07992=1124.961,305.777,-76.888,-177.844,10.503,149.533
C07993=1124.966,305.529,-76.856,-177.847,10.501,149.533
C07994=1124.970,305.281,-76.824,-177.850,10.498,149.533
C07995=1124.974,305.033,-76.792,-177.853,10.495,149.533
C07996=1124.978,304.785,-76.760,-177.857,10.493,149.534
C07997=1124.982,304.537,-76.728,-177.859,10.490,149.534
C07998=1124.986,304.290,-76.697,-177.863,10.488,149.534
C07999=1124.990,304.042,-76.664,-177.866,10.485,149.534
C08000=1124.994,303.794,-76.632,-177.869,10.483,149.534
C08001=1124.998,303.547,-76.600,-177.872,10.480,149.534
C08002=1125.003,303.298,-76.568,-177.875,10.478,149.535
C08003=1125.007,303.050,-76.537,-177.878,10.475,149.535
C08004=1125.011,302.802,-76.505,-177.881,10.473,149.535
C08005=1125.015,302.554,-76.473,-177.884,10.470,149.535
C08006=1125.019,302.306,-76.441,-177.887,10.468,149.535
C08007=1125.024,302.058,-76.409,-177.891,10.465,149.536
C08008=1125.027,301.810,-76.378,-177.894,10.463,149.536
C08009=1125.031,301.562,-76.346,-177.897,10.460,149.536
C08010=1125.036,301.315,-76.314,-177.900,10.457,149.536
C08011=1125.040,301.067,-76.282,-177.903,10.455,149.536
C08012=1125.043,300.819,-76.250,-177.906,10.452,149.536
C08013=1125.048,300.571,-76.219,-177.909,10.450,149.537
C08014=1125.052,300.323,-76.187,-177.912,10.447,149.537
C08015=1125.056,300.074,-76.155,-177.915,10.445,149.537
C08016=1125.061,299.827,-76.123,-177.918,10.443,149.537
C08017=1125.064,299.579,-76.092,-177.921,10.440,149.537
C08018=1125.069,299.331,-76.061,-177.924,10.437,149.537
C08019=1125.073,299.083,-76.029,-177.928,10.435,149.538
C08020=1125.076,298.835,-75.997,-177.930,10.432,149.538
C08021=1125.081,298.588,-75.966,-177.934,10.430,149.538
C08022=1125.085,298.339,-75.934,-177.937,10.427,149.538
C08023=1125.090,298.091,-75.902,-177.940,10.425,149.538
C08024=1125.093,297.843,-75.871,-177.943,10.422,149.538
C08025=1125.097,297.595,-75.839,-177.946,10.419,149.539
C08026=1125.102,297.347,-75.808,-177.949,10.417,149.539
C08027=1125.105,297.099,-75.776,-177.952,10.415,149.539
C08028=1125.110,296.851,-75.745,-177.955,10.412,149.539
C08029=1125.114,296.603,-75.713,-177.958,10.410,149.539
C08030=1125.118,296.355,-75.683,-177.961,10.407,149.540
C08031=1125.122,296.107,-75.651,-177.965,10.405,149.540
C08032=1125.126,295.860,-75.619,-177.967,10.402,149.540
C08033=1125.130,295.611,-75.588,-177.971,10.399,149.540
C08034=1125.135,295.364,-75.557,-177.974,10.397,149.540
C08035=1125.139,295.115,-75.526,-177.977,10.394,149.541
C08036=1125.142,294.902,-75.498,-177.979,10.392,149.541
C08037=1125.146,294.689,-75.472,-177.982,10.390,149.541
C08038=1125.150,294.476,-75.445,-177.985,10.387,149.541
C08039=1125.153,294.263,-75.418,-177.987,10.386,149.541
C08040=1125.157,294.049,-75.391,-177.990,10.383,149.541
C08041=1125.159,293.836,-75.365,-177.993,10.381,149.541
C08042=1125.163,293.623,-75.338,-177.995,10.379,149.541
C08043=1125.167,293.410,-75.311,-177.998,10.377,149.542
C08044=1125.171,293.162,-75.280,-178.001,10.374,149.542
C08045=1125.175,292.914,-75.248,-178.004,10.372,149.542
C08046=1125.179,292.666,-75.217,-178.007,10.369,149.542
C08047=1125.183,292.418,-75.185,-178.010,10.367,149.542
C08048=1125.188,292.170,-75.155,-178.013,10.364,149.543
C08049=1125.192,291.921,-75.124,-178.016,10.362,149.543
C08050=1125.195,291.674,-75.093,-178.019,10.359,149.543
C08051=1125.199,291.425,-75.062,-178.022,10.356,149.543
C08052=1125.204,291.177,-75.031,-178.026,10.354,149.543
C08053=1125.208,290.930,-74.999,-178.029,10.351,149.543
C08054=1125.212,290.681,-74.968,-178.032,10.349,149.544
C08055=1125.217,290.433,-74.937,-178.034,10.347,149.544
C08056=1125.220,290.185,-74.907,-178.038,10.344,149.544
C08057=1125.225,289.938,-74.875,-178.040,10.341,149.544
C08058=1125.229,289.689,-74.844,-178.044,10.339,149.544
C08059=1125.233,289.441,-74.814,-178.047,10.336,149.545
C08060=1125.238,289.193,-74.783,-178.050,10.334,149.545
C08061=1125.241,288.945,-74.752,-178.053,10.331,149.545
C08062=1125.245,288.698,-74.721,-178.056,10.329,149.545
C08063=1125.249,288.449,-74.690,-178.059,10.326,149.545
C08064=1125.254,288.201,-74.659,-178.062,10.323,149.545
C08065=1125.258,287.953,-74.629,-178.066,10.321,149.546
C08066=1125.262,287.705,-74.598,-178.068,10.319,149.546
C08067=1125.266,287.457,-74.567,-178.071,10.316,149.546
C08068=1125.270,287.209,-74.537,-178.074,10.314,149.546
C08069=1125.274,286.960,-74.506,-178.077,10.311,149.546
C08070=1125.279,286.712,-74.475,-178.080,10.308,149.546
C08071=1125.284,286.464,-74.444,-178.084,10.306,149.547
C08072=1125.287,286.216,-74.413,-178.087,10.303,149.547
C08073=1125.291,285.969,-74.382,-178.090,10.300,149.547
C08074=1125.295,285.720,-74.353,-178.093,10.298,149.547
C08075=1125.299,285.472,-74.321,-178.096,10.295,149.547
C08076=1125.304,285.224,-74.291,-178.099,10.294,149.548
C08077=1125.308,284.976,-74.260,-178.102,10.291,149.548
C08078=1125.312,284.728,-74.229,-178.105,10.288,149.548
C08079=1125.316,284.480,-74.199,-178.108,10.286,149.548
C08080=1125.320,284.232,-74.168,-178.111,10.283,149.548
C08081=1125.325,283.984,-74.138,-178.114,10.280,149.548
C08082=1125.328,283.736,-74.107,-178.117,10.278,149.549
C08083=1125.333,283.488,-74.076,-178.120,10.275,149.549
C08084=1125.337,283.240,-74.046,-178.123,10.273,149.549
C08085=1125.341,282.992,-74.015,-178.127,10.270,149.549
C08086=1125.346,282.743,-73.985,-178.129,10.268,149.549
C08087=1125.350,282.495,-73.955,-178.132,10.265,149.549
C08088=1125.354,282.247,-73.924,-178.135,10.263,149.550
C08089=1125.358,282.000,-73.894,-178.138,10.260,149.550
C08090=1125.362,281.751,-73.863,-178.142,10.258,149.550
C08091=1125.366,281.503,-73.833,-178.144,10.255,149.550
C08092=1125.370,281.289,-73.807,-178.148,10.253,149.550
C08093=1125.373,281.077,-73.781,-178.150,10.251,149.551
C08094=1125.377,280.862,-73.755,-178.153,10.248,149.551
C08095=1125.381,280.649,-73.728,-178.156,10.245,149.551
C08096=1125.384,280.436,-73.702,-178.159,10.243,149.551
C08097=1125.389,280.223,-73.677,-178.162,10.241,149.551
C08098=1125.391,280.009,-73.650,-178.165,10.238,149.551
C08099=1125.395,279.796,-73.624,-178.168,10.236,149.552
C08100=1125.400,279.548,-73.594,-178.171,10.233,149.552
C08101=1125.404,279.300,-73.564,-178.175,10.231,149.552
C08102=1125.408,279.051,-73.534,-178.178,10.227,149.552
C08103=1125.412,278.804,-73.504,-178.182,10.225,149.552
C08104=1125.416,278.555,-73.473,-178.184,10.222,149.553
C08105=1125.420,278.307,-73.443,-178.188,10.220,149.553
C08106=1125.424,278.059,-73.413,-178.191,10.217,149.553
C08107=1125.429,277.811,-73.383,-178.195,10.214,149.553
C08108=1125.433,277.563,-73.353,-178.198,10.211,149.553
C08109=1125.437,277.315,-73.324,-178.201,10.208,149.553
C08110=1125.441,277.066,-73.292,-178.204,10.206,149.554
C08111=1125.445,276.818,-73.263,-178.207,10.203,149.554
C08112=1125.449,276.570,-73.233,-178.210,10.200,149.554
C08113=1125.454,276.322,-73.203,-178.214,10.197,149.554
C08114=1125.458,276.074,-73.173,-178.217,10.194,149.554
C08115=1125.462,275.826,-73.143,-178.220,10.191,149.554
C08116=1125.466,275.578,-73.113,-178.223,10.189,149.555
C08117=1125.471,275.329,-73.083,-178.226,10.186,149.555
C08118=1125.475,275.081,-73.053,-178.229,10.184,149.555
C08119=1125.479,274.834,-73.023,-178.232,10.181,149.555
C08120=1125.483,274.585,-72.994,-178.235,10.178,149.555
C08121=1125.488,274.336,-72.963,-178.238,10.176,149.555
C08122=1125.492,274.088,-72.933,-178.241,10.173,149.555
C08123=1125.496,273.840,-72.904,-178.244,10.170,149.556
C08124=1125.500,273.592,-72.874,-178.247,10.167,149.556
C08125=1125.505,273.344,-72.844,-178.250,10.165,149.556
C08126=1125.509,273.096,-72.814,-178.253,10.162,149.556
C08127=1125.513,272.847,-72.785,-178.256,10.159,149.556
C08128=1125.517,272.599,-72.755,-178.259,10.157,149.556
C08129=1125.521,272.351,-72.725,-178.262,10.154,149.556
C08130=1125.525,272.103,-72.696,-178.265,10.151,149.556
C08131=1125.530,271.855,-72.666,-178.267,10.149,149.557
C08132=1125.534,271.606,-72.636,-178.270,10.146,149.557
C08133=1125.538,271.358,-72.607,-178.273,10.144,149.557
C08134=1125.543,271.110,-72.577,-178.276,10.141,149.557
C08135=1125.546,270.862,-72.547,-178.279,10.138,149.557
C08136=1125.551,270.614,-72.518,-178.282,10.135,149.557
C08137=1125.555,270.366,-72.488,-178.284,10.133,149.557
C08138=1125.559,270.117,-72.459,-178.287,10.131,149.557
C08139=1125.563,269.869,-72.429,-178.290,10.128,149.557
C08140=1125.567,269.621,-72.400,-178.293,10.125,149.557
C08141=1125.572,269.373,-72.370,-178.295,10.123,149.558
C08142=1125.576,269.124,-72.340,-178.298,10.120,149.558
C08143=1125.581,268.876,-72.311,-178.301,10.118,149.558
C08144=1125.585,268.628,-72.282,-178.304,10.116,149.558
C08145=1125.590,268.380,-72.252,-178.307,10.113,149.558
C08146=1125.594,268.132,-72.223,-178.309,10.110,149.558
C08147=1125.598,267.883,-72.193,-178.312,10.108,149.558
C08148=1125.602,267.670,-72.168,-178.314,10.106,149.558
C08149=1125.605,267.456,-72.143,-178.316,10.104,149.559
C08150=1125.609,267.243,-72.118,-178.318,10.102,149.558
C08151=1125.612,267.030,-72.093,-178.321,10.100,149.559
C08152=1125.616,266.816,-72.067,-178.324,10.097,149.559
C08153=1125.619,266.603,-72.042,-178.326,10.095,149.559
C08154=1125.624,266.389,-72.017,-178.328,10.093,149.559
C08155=1125.627,266.176,-71.991,-178.330,10.091,149.559
C08156=1125.631,265.927,-71.962,-178.332,10.089,149.559
C08157=1125.636,265.679,-71.932,-178.335,10.086,149.559
C08158=1125.640,265.431,-71.903,-178.338,10.084,149.559
C08159=1125.643,265.183,-71.874,-178.340,10.082,149.559
C08160=1125.648,264.934,-71.845,-178.343,10.079,149.559
C08161=1125.652,264.686,-71.816,-178.345,10.077,149.560
C08162=1125.657,264.438,-71.787,-178.348,10.075,149.560
C08163=1125.661,264.190,-71.757,-178.352,10.071,149.560
C08164=1125.665,263.942,-71.728,-178.355,10.069,149.560
C08165=1125.670,263.693,-71.699,-178.359,10.065,149.560
C08166=1125.674,263.444,-71.670,-178.363,10.062,149.561
C08167=1125.678,263.196,-71.640,-178.366,10.060,149.561
C08168=1125.683,262.949,-71.611,-178.370,10.056,149.561
C08169=1125.686,262.700,-71.583,-178.373,10.053,149.561
C08170=1125.691,262.452,-71.554,-178.377,10.050,149.561
C08171=1125.695,262.204,-71.524,-178.380,10.047,149.562
C08172=1125.699,261.955,-71.495,-178.384,10.044,149.562
C08173=1125.704,261.707,-71.466,-178.387,10.041,149.562
C08174=1125.707,261.459,-71.437,-178.391,10.039,149.562
C08175=1125.712,261.210,-71.409,-178.394,10.035,149.562
C08176=1125.716,260.962,-71.379,-178.397,10.032,149.562
C08177=1125.721,260.714,-71.351,-178.401,10.029,149.563
C08178=1125.725,260.466,-71.322,-178.404,10.026,149.563
C08179=1125.729,260.217,-71.293,-178.408,10.023,149.563
C08180=1125.733,259.969,-71.264,-178.411,10.020,149.563
C08181=1125.738,259.721,-71.235,-178.414,10.017,149.563
C08182=1125.742,259.473,-71.207,-178.417,10.014,149.563
C08183=1125.746,259.224,-71.178,-178.421,10.011,149.563
C08184=1125.751,258.975,-71.148,-178.423,10.009,149.564
C08185=1125.755,258.728,-71.121,-178.426,10.006,149.564
C08186=1125.759,258.479,-71.091,-178.430,10.002,149.564
C08187=1125.764,258.230,-71.062,-178.433,10.000,149.564
C08188=1125.768,257.983,-71.034,-178.436,9.997,149.564
C08189=1125.772,257.734,-71.005,-178.439,9.994,149.564
C08190=1125.776,257.486,-70.977,-178.441,9.991,149.564
C08191=1125.780,257.237,-70.948,-178.444,9.988,149.564
C08192=1125.785,256.989,-70.919,-178.447,9.985,149.564
C08193=1125.789,256.741,-70.890,-178.450,9.983,149.564
C08194=1125.793,256.492,-70.862,-178.453,9.980,149.564
C08195=1125.797,256.244,-70.834,-178.456,9.977,149.565
C08196=1125.802,255.996,-70.805,-178.459,9.974,149.565
C08197=1125.806,255.747,-70.776,-178.459,9.973,149.564
C08198=1125.810,255.499,-70.748,-178.459,9.972,149.564
C08199=1125.815,255.251,-70.719,-178.459,9.971,149.564
C08200=1125.819,255.003,-70.691,-178.459,9.970,149.564
C08201=1125.823,254.754,-70.662,-178.460,9.968,149.563
C08202=1125.827,254.506,-70.634,-178.461,9.967,149.563
C08203=1125.832,254.258,-70.605,-178.462,9.965,149.563
C08204=1125.836,254.044,-70.580,-178.462,9.964,149.563
C08205=1125.840,253.830,-70.556,-178.464,9.963,149.563
C08206=1125.843,253.617,-70.531,-178.465,9.961,149.563
C08207=1125.846,253.403,-70.507,-178.467,9.960,149.563
C08208=1125.851,253.190,-70.483,-178.469,9.957,149.563
C08209=1125.854,252.976,-70.457,-178.470,9.956,149.563
C08210=1125.858,252.763,-70.434,-178.472,9.954,149.563
C08211=1125.861,252.548,-70.409,-178.474,9.952,149.563
C08212=1125.866,252.301,-70.381,-178.477,9.950,149.564
C08213=1125.870,252.052,-70.352,-178.480,9.948,149.564
C08214=1125.874,251.804,-70.324,-178.483,9.945,149.564
C08215=1125.879,251.556,-70.295,-178.486,9.942,149.564
C08216=1125.883,251.307,-70.267,-178.489,9.940,149.564
C08217=1125.888,251.059,-70.239,-178.493,9.937,149.565
C08218=1125.891,250.811,-70.210,-178.497,9.933,149.565
C08219=1125.896,250.562,-70.181,-178.501,9.930,149.565
C08220=1125.900,250.314,-70.153,-178.506,9.927,149.566
C08221=1125.904,250.065,-70.125,-178.510,9.923,149.566
C08222=1125.909,249.817,-70.097,-178.515,9.919,149.566
C08223=1125.913,249.569,-70.069,-178.520,9.916,149.567
C08224=1125.918,249.321,-70.040,-178.526,9.912,149.567
C08225=1125.921,249.072,-70.012,-178.530,9.908,149.567
C08226=1125.926,248.824,-69.985,-178.536,9.903,149.568
C08227=1125.930,248.575,-69.956,-178.542,9.899,149.568
C08228=1125.935,248.327,-69.928,-178.548,9.894,149.569
C08229=1125.939,248.078,-69.901,-178.554,9.889,149.569
C08230=1125.944,247.830,-69.872,-178.560,9.885,149.570
C08231=1125.947,247.581,-69.844,-178.567,9.879,149.570
C08232=1125.952,247.334,-69.816,-178.571,9.875,149.570
C08233=1125.956,247.085,-69.788,-178.573,9.873,149.570
C08234=1125.961,246.836,-69.761,-178.574,9.871,149.570
C08235=1125.965,246.588,-69.732,-178.575,9.869,149.570
C08236=1125.969,246.340,-69.705,-178.577,9.866,149.570
C08237=1125.973,246.092,-69.677,-178.578,9.864,149.570
C08238=1125.977,245.843,-69.649,-178.580,9.862,149.569
C08239=1125.983,245.594,-69.621,-178.582,9.859,149.569
C08240=1125.986,245.346,-69.593,-178.583,9.858,149.569
C08241=1125.991,245.097,-69.566,-178.585,9.855,149.569
C08242=1125.995,244.849,-69.538,-178.586,9.853,149.569
C08243=1125.999,244.601,-69.510,-178.588,9.850,149.569
C08244=1126.004,244.352,-69.482,-178.590,9.848,149.569
C08245=1126.008,244.104,-69.454,-178.591,9.846,149.569
C08246=1126.013,243.856,-69.426,-178.593,9.844,149.569
C08247=1126.017,243.607,-69.399,-178.595,9.842,149.569
C08248=1126.021,243.359,-69.371,-178.597,9.839,149.569
C08249=1126.025,243.111,-69.343,-178.599,9.837,149.569
C08250=1126.029,242.861,-69.316,-178.601,9.835,149.569
C08251=1126.034,242.613,-69.288,-178.603,9.833,149.569
C08252=1126.039,242.365,-69.260,-178.605,9.830,149.569
C08253=1126.043,242.116,-69.232,-178.607,9.828,149.569
C08254=1126.047,241.868,-69.205,-178.609,9.825,149.569
C08255=1126.051,241.619,-69.177,-178.612,9.823,149.569
C08256=1126.056,241.371,-69.149,-178.614,9.821,149.569
C08257=1126.060,241.123,-69.122,-178.615,9.818,149.569
C08258=1126.064,240.874,-69.094,-178.618,9.816,149.569
C08259=1126.069,240.626,-69.067,-178.620,9.813,149.569
C08260=1126.073,240.412,-69.043,-178.623,9.811,149.569
C08261=1126.076,240.199,-69.019,-178.624,9.810,149.569
C08262=1126.079,239.985,-68.995,-178.626,9.807,149.569
C08263=1126.084,239.771,-68.972,-178.628,9.805,149.569
C08264=1126.087,239.557,-68.948,-178.630,9.803,149.569
C08265=1126.091,239.344,-68.924,-178.632,9.801,149.569
C08266=1126.095,239.130,-68.901,-178.634,9.799,149.569
C08267=1126.099,238.917,-68.877,-178.637,9.797,149.569
C08268=1126.103,238.667,-68.850,-178.639,9.794,149.569
C08269=1126.107,238.419,-68.822,-178.641,9.792,149.569
C08270=1126.112,238.171,-68.795,-178.644,9.789,149.569
C08271=1126.116,237.922,-68.767,-178.647,9.787,149.569
C08272=1126.120,237.674,-68.740,-178.650,9.784,149.569
C08273=1126.125,237.425,-68.713,-178.652,9.781,149.569
C08274=1126.129,237.177,-68.685,-178.655,9.778,149.570
C08275=1126.134,236.928,-68.657,-178.657,9.777,149.570
C08276=1126.138,236.680,-68.630,-178.660,9.774,149.570
C08277=1126.143,236.432,-68.603,-178.663,9.771,149.570
C08278=1126.147,236.183,-68.575,-178.666,9.768,149.570
C08279=1126.151,235.934,-68.548,-178.669,9.766,149.570
C08280=1126.156,235.686,-68.520,-178.672,9.763,149.570
C08281=1126.160,235.438,-68.493,-178.675,9.760,149.570
C08282=1126.164,235.189,-68.466,-178.678,9.757,149.570
C08283=1126.168,234.940,-68.439,-178.681,9.754,149.570
C08284=1126.173,234.693,-68.412,-178.683,9.751,149.571
C08285=1126.177,234.444,-68.385,-178.686,9.749,149.571
C08286=1126.182,234.196,-68.358,-178.689,9.746,149.571
C08287=1126.186,233.946,-68.330,-178.692,9.743,149.571
C08288=1126.191,233.698,-68.303,-178.695,9.740,149.571
C08289=1126.195,233.450,-68.277,-178.699,9.737,149.571
C08290=1126.199,233.202,-68.249,-178.702,9.735,149.572
C08291=1126.204,232.953,-68.222,-178.705,9.732,149.572
C08292=1126.208,232.704,-68.194,-178.709,9.728,149.572
C08293=1126.212,232.456,-68.167,-178.712,9.726,149.572
C08294=1126.216,232.207,-68.141,-178.715,9.722,149.572
C08295=1126.221,231.959,-68.114,-178.718,9.719,149.572
C08296=1126.225,231.710,-68.087,-178.722,9.716,149.572
C08297=1126.230,231.462,-68.060,-178.725,9.713,149.572
C08298=1126.233,231.213,-68.033,-178.728,9.709,149.572
C08299=1126.238,230.965,-68.006,-178.731,9.707,149.573
C08300=1126.243,230.716,-67.979,-178.735,9.704,149.573
C08301=1126.247,230.468,-67.952,-178.739,9.700,149.573
C08302=1126.251,230.219,-67.925,-178.742,9.696,149.573
C08303=1126.256,229.971,-67.898,-178.746,9.693,149.573
C08304=1126.261,229.722,-67.871,-178.750,9.689,149.573
C08305=1126.265,229.474,-67.845,-178.753,9.687,149.574
C08306=1126.269,229.226,-67.817,-178.756,9.683,149.574
C08307=1126.274,228.977,-67.790,-178.760,9.680,149.574
C08308=1126.278,228.728,-67.765,-178.763,9.676,149.574
C08309=1126.282,228.479,-67.737,-178.767,9.673,149.574
C08310=1126.286,228.231,-67.711,-178.770,9.669,149.574
C08311=1126.291,227.983,-67.684,-178.773,9.666,149.574
C08312=1126.295,227.734,-67.657,-178.777,9.663,149.574
C08313=1126.300,227.485,-67.631,-178.781,9.659,149.574
C08314=1126.304,227.237,-67.604,-178.784,9.657,149.575
C08315=1126.308,226.989,-67.577,-178.787,9.653,149.574
C08316=1126.312,226.775,-67.555,-178.790,9.650,149.575
C08317=1126.316,226.561,-67.532,-178.792,9.647,149.575
C08318=1126.320,226.347,-67.509,-178.795,9.644,149.575
C08319=1126.324,226.133,-67.486,-178.798,9.641,149.575
C08320=1126.328,225.920,-67.463,-178.801,9.638,149.575
C08321=1126.331,225.705,-67.440,-178.803,9.635,149.575
C08322=1126.335,225.492,-67.417,-178.806,9.632,149.575
C08323=1126.339,225.278,-67.394,-178.809,9.629,149.575
C08324=1126.344,225.029,-67.369,-178.812,9.627,149.575
C08325=1126.348,224.781,-67.341,-178.815,9.623,149.575
C08326=1126.352,224.533,-67.315,-178.818,9.620,149.575
C08327=1126.356,224.284,-67.289,-178.821,9.616,149.575
C08328=1126.361,224.035,-67.262,-178.823,9.613,149.575
C08329=1126.365,223.786,-67.236,-178.826,9.610,149.575
C08330=1126.370,223.538,-67.209,-178.829,9.606,149.575
C08331=1126.374,223.289,-67.184,-178.832,9.603,149.575
C08332=1126.379,223.041,-67.157,-178.834,9.600,149.575
C08333=1126.383,222.792,-67.131,-178.838,9.596,149.575
C08334=1126.387,222.544,-67.104,-178.841,9.593,149.575
C08335=1126.392,222.295,-67.078,-178.843,9.590,149.575
C08336=1126.396,222.046,-67.052,-178.846,9.587,149.575
C08337=1126.401,221.798,-67.026,-178.848,9.584,149.575
C08338=1126.406,221.549,-67.000,-178.851,9.580,149.575
C08339=1126.409,221.301,-66.973,-178.854,9.577,149.574
C08340=1126.414,221.052,-66.947,-178.856,9.574,149.574
C08341=1126.418,220.804,-66.921,-178.859,9.571,149.574
C08342=1126.423,220.555,-66.895,-178.861,9.568,149.574
C08343=1126.427,220.306,-66.869,-178.864,9.565,149.574
C08344=1126.431,220.058,-66.842,-178.867,9.562,149.574
C08345=1126.436,219.809,-66.817,-178.869,9.558,149.574
C08346=1126.441,219.561,-66.791,-178.872,9.555,149.574
C08347=1126.445,219.311,-66.765,-178.874,9.552,149.574
C08348=1126.449,219.063,-66.738,-178.876,9.549,149.574
C08349=1126.454,218.815,-66.712,-178.878,9.546,149.574
C08350=1126.458,218.566,-66.687,-178.881,9.543,149.574
C08351=1126.463,218.318,-66.660,-178.883,9.540,149.574
C08352=1126.467,218.069,-66.634,-178.885,9.537,149.573
C08353=1126.472,217.820,-66.608,-178.888,9.534,149.573
C08354=1126.476,217.571,-66.583,-178.890,9.531,149.573
C08355=1126.480,217.323,-66.557,-178.892,9.528,149.573
C08356=1126.485,217.074,-66.530,-178.894,9.525,149.573
C08357=1126.490,216.826,-66.504,-178.896,9.522,149.573
C08358=1126.494,216.577,-66.479,-178.899,9.519,149.573
C08359=1126.498,216.328,-66.453,-178.900,9.517,149.572
C08360=1126.502,216.080,-66.427,-178.903,9.513,149.572
C08361=1126.507,215.832,-66.402,-178.904,9.511,149.572
C08362=1126.512,215.582,-66.375,-178.907,9.508,149.572
C08363=1126.516,215.334,-66.349,-178.909,9.505,149.572
C08364=1126.520,215.085,-66.323,-178.911,9.502,149.572
C08365=1126.524,214.837,-66.297,-178.913,9.500,149.572
C08366=1126.529,214.589,-66.272,-178.915,9.496,149.571
C08367=1126.533,214.340,-66.246,-178.917,9.494,149.571
C08368=1126.538,214.091,-66.221,-178.918,9.491,149.571
C08369=1126.542,213.842,-66.195,-178.920,9.489,149.571
C08370=1126.547,213.594,-66.169,-178.923,9.486,149.571
C08371=1126.552,213.345,-66.143,-178.924,9.483,149.571
C08372=1126.555,213.131,-66.122,-178.926,9.481,149.571
C08373=1126.559,212.917,-66.099,-178.927,9.479,149.571
C08374=1126.563,212.703,-66.077,-178.929,9.476,149.571
C08375=1126.567,212.490,-66.055,-178.930,9.474,149.570
C08376=1126.570,212.275,-66.033,-178.932,9.471,149.570
C08377=1126.574,212.061,-66.011,-178.933,9.470,149.570
C08378=1126.578,211.847,-65.988,-178.935,9.467,149.570
C08379=1126.582,211.633,-65.966,-178.937,9.465,149.570
C08380=1126.586,211.384,-65.941,-178.938,9.462,149.570
C08381=1126.591,211.136,-65.915,-178.941,9.459,149.570
C08382=1126.595,210.887,-65.889,-178.943,9.457,149.570
C08383=1126.599,210.639,-65.864,-178.945,9.455,149.570
C08384=1126.605,210.390,-65.839,-178.947,9.451,149.570
C08385=1126.609,210.141,-65.813,-178.949,9.449,149.570
C08386=1126.613,209.892,-65.788,-178.952,9.446,149.570
C08387=1126.618,209.644,-65.762,-178.954,9.444,149.570
C08388=1126.622,209.395,-65.736,-178.957,9.441,149.570
C08389=1126.626,209.147,-65.711,-178.958,9.439,149.570
C08390=1126.631,208.898,-65.685,-178.961,9.436,149.570
C08391=1126.636,208.649,-65.660,-178.963,9.434,149.570
C08392=1126.640,208.400,-65.634,-178.966,9.430,149.570
C08393=1126.645,208.152,-65.609,-178.968,9.427,149.570
C08394=1126.649,207.903,-65.583,-178.971,9.425,149.570
C08395=1126.654,207.655,-65.558,-178.973,9.422,149.570
C08396=1126.658,207.406,-65.533,-178.976,9.420,149.570
C08397=1126.663,207.157,-65.507,-178.979,9.416,149.570
C08398=1126.667,206.909,-65.482,-178.981,9.414,149.570
C08399=1126.671,206.660,-65.457,-178.984,9.411,149.570
C08400=1126.676,206.412,-65.432,-178.987,9.409,149.570
C08401=1126.680,206.163,-65.406,-178.989,9.406,149.570
C08402=1126.684,205.914,-65.380,-178.992,9.403,149.570
C08403=1126.690,205.665,-65.356,-178.995,9.400,149.570
C08404=1126.694,205.417,-65.330,-178.997,9.397,149.570
C08405=1126.699,205.168,-65.305,-179.000,9.394,149.570
C08406=1126.702,204.919,-65.280,-179.003,9.391,149.571
C08407=1126.707,204.671,-65.255,-179.006,9.389,149.571
C08408=1126.712,204.422,-65.230,-179.009,9.386,149.571
C08409=1126.716,204.173,-65.204,-179.012,9.383,149.571
C08410=1126.721,203.924,-65.179,-179.015,9.380,149.571
C08411=1126.725,203.676,-65.154,-179.018,9.377,149.571
C08412=1126.730,203.427,-65.130,-179.021,9.374,149.571
C08413=1126.734,203.178,-65.104,-179.024,9.371,149.571
C08414=1126.739,202.930,-65.078,-179.028,9.368,149.571
C08415=1126.743,202.681,-65.054,-179.030,9.364,149.571
C08416=1126.747,202.433,-65.029,-179.033,9.362,149.572
C08417=1126.752,202.184,-65.004,-179.037,9.358,149.572
C08418=1126.757,201.935,-64.979,-179.040,9.355,149.572
C08419=1126.761,201.686,-64.954,-179.043,9.352,149.572
C08420=1126.766,201.438,-64.929,-179.046,9.349,149.572
C08421=1126.770,201.189,-64.903,-179.050,9.346,149.572
C08422=1126.774,200.940,-64.879,-179.053,9.343,149.572
C08423=1126.779,200.691,-64.854,-179.056,9.339,149.573
C08424=1126.784,200.443,-64.829,-179.060,9.336,149.573
C08425=1126.787,200.194,-64.804,-179.064,9.332,149.573
C08426=1126.793,199.945,-64.780,-179.067,9.330,149.573
C08427=1126.797,199.696,-64.754,-179.070,9.326,149.573
C08428=1126.801,199.482,-64.734,-179.073,9.323,149.573
C08429=1126.805,199.268,-64.712,-179.077,9.320,149.573
C08430=1126.809,199.054,-64.691,-179.079,9.317,149.573
C08431=1126.812,198.840,-64.669,-179.082,9.314,149.574
C08432=1126.816,198.626,-64.648,-179.085,9.311,149.574
C08433=1126.820,198.412,-64.627,-179.089,9.308,149.574
C08434=1126.823,198.198,-64.605,-179.092,9.305,149.574
C08435=1126.828,197.983,-64.584,-179.095,9.302,149.574
C08436=1126.832,197.735,-64.559,-179.099,9.298,149.574
C08437=1126.837,197.487,-64.535,-179.102,9.294,149.574
C08438=1126.841,197.237,-64.510,-179.106,9.291,149.574
C08439=1126.846,196.989,-64.485,-179.109,9.287,149.574
C08440=1126.850,196.740,-64.461,-179.113,9.283,149.575
C08441=1126.855,196.491,-64.436,-179.117,9.279,149.575
C08442=1126.859,196.242,-64.412,-179.121,9.276,149.575
C08443=1126.865,195.994,-64.388,-179.122,9.273,149.575
C08444=1126.868,195.745,-64.363,-179.124,9.270,149.574
C08445=1126.873,195.496,-64.339,-179.125,9.268,149.574
C08446=1126.878,195.247,-64.314,-179.127,9.265,149.574
C08447=1126.882,194.998,-64.290,-179.128,9.263,149.574
C08448=1126.887,194.750,-64.265,-179.130,9.260,149.574
C08449=1126.891,194.501,-64.241,-179.132,9.258,149.574
C08450=1126.896,194.252,-64.216,-179.134,9.255,149.574
C08451=1126.900,194.003,-64.192,-179.135,9.253,149.573
C08452=1126.904,193.755,-64.168,-179.137,9.250,149.573
C08453=1126.910,193.506,-64.143,-179.138,9.248,149.573
C08454=1126.913,193.257,-64.119,-179.140,9.245,149.573
C08455=1126.919,193.008,-64.094,-179.142,9.243,149.573
C08456=1126.923,192.760,-64.070,-179.144,9.239,149.573
C08457=1126.927,192.511,-64.046,-179.146,9.237,149.573
C08458=1126.932,192.262,-64.021,-179.148,9.235,149.573
C08459=1126.936,192.014,-63.997,-179.150,9.232,149.572
C08460=1126.941,191.765,-63.973,-179.152,9.229,149.572
C08461=1126.945,191.516,-63.948,-179.154,9.227,149.572
C08462=1126.950,191.267,-63.925,-179.156,9.224,149.572
C08463=1126.954,191.018,-63.900,-179.157,9.222,149.572
C08464=1126.959,190.770,-63.876,-179.160,9.219,149.572
C08465=1126.963,190.521,-63.851,-179.162,9.216,149.572
C08466=1126.968,190.272,-63.827,-179.164,9.213,149.572
C08467=1126.973,190.023,-63.803,-179.166,9.211,149.572
C08468=1126.977,189.774,-63.779,-179.169,9.208,149.572
C08469=1126.982,189.526,-63.755,-179.171,9.205,149.572
C08470=1126.986,189.277,-63.730,-179.173,9.202,149.572
C08471=1126.991,189.028,-63.706,-179.175,9.200,149.572
C08472=1126.995,188.779,-63.683,-179.177,9.196,149.572
C08473=1127.000,188.531,-63.659,-179.179,9.194,149.571
C08474=1127.005,188.282,-63.634,-179.182,9.191,149.571
C08475=1127.009,188.033,-63.610,-179.183,9.189,149.571
C08476=1127.013,187.784,-63.586,-179.186,9.186,149.571
C08477=1127.018,187.535,-63.562,-179.189,9.183,149.572
C08478=1127.023,187.287,-63.537,-179.191,9.180,149.571
C08479=1127.028,187.038,-63.514,-179.193,9.177,149.571
C08480=1127.031,186.789,-63.490,-179.196,9.174,149.571
C08481=1127.036,186.540,-63.466,-179.198,9.171,149.571
C08482=1127.041,186.291,-63.442,-179.201,9.168,149.571
C08483=1127.046,186.042,-63.418,-179.203,9.166,149.571
C08484=1127.049,185.828,-63.397,-179.205,9.163,149.571
C08485=1127.053,185.614,-63.377,-179.207,9.160,149.571
C08486=1127.057,185.400,-63.356,-179.210,9.158,149.571
C08487=1127.061,185.185,-63.335,-179.212,9.155,149.571
C08488=1127.065,184.972,-63.316,-179.214,9.153,149.571
C08489=1127.069,184.758,-63.294,-179.217,9.150,149.571
C08490=1127.073,184.543,-63.273,-179.218,9.147,149.571
C08491=1127.077,184.329,-63.253,-179.220,9.145,149.571
C08492=1127.082,184.080,-63.230,-179.223,9.142,149.571
C08493=1127.086,183.831,-63.205,-179.226,9.138,149.571
C08494=1127.090,183.582,-63.182,-179.229,9.135,149.571
C08495=1127.095,183.334,-63.158,-179.231,9.132,149.571
C08496=1127.099,183.085,-63.134,-179.234,9.130,149.571
C08497=1127.104,182.836,-63.110,-179.237,9.126,149.571
C08498=1127.108,182.587,-63.087,-179.239,9.123,149.571
C08499=1127.113,182.338,-63.064,-179.243,9.119,149.571
C08500=1127.117,182.090,-63.040,-179.246,9.117,149.571
C08501=1127.122,181.841,-63.016,-179.248,9.114,149.571
C08502=1127.127,181.592,-62.992,-179.251,9.110,149.571
C08503=1127.131,181.343,-62.969,-179.254,9.107,149.571
C08504=1127.136,181.094,-62.945,-179.257,9.104,149.571
C08505=1127.140,180.846,-62.921,-179.259,9.101,149.571
C08506=1127.145,180.597,-62.898,-179.262,9.097,149.571
C08507=1127.150,180.348,-62.875,-179.265,9.094,149.572
C08508=1127.154,180.099,-62.851,-179.269,9.090,149.571
C08509=1127.159,179.850,-62.827,-179.271,9.087,149.571
C08510=1127.164,179.601,-62.804,-179.275,9.084,149.572
C08511=1127.168,179.353,-62.780,-179.278,9.080,149.572
C08512=1127.173,179.104,-62.756,-179.280,9.077,149.571
C08513=1127.177,178.855,-62.733,-179.282,9.074,149.571
C08514=1127.182,178.606,-62.710,-179.284,9.071,149.571
C08515=1127.187,178.357,-62.686,-179.286,9.068,149.571
C08516=1127.190,178.109,-62.663,-179.288,9.065,149.571
C08517=1127.195,177.859,-62.639,-179.291,9.062,149.571
C08518=1127.200,177.610,-62.616,-179.293,9.060,149.571
C08519=1127.205,177.361,-62.593,-179.295,9.056,149.571
C08520=1127.209,177.112,-62.569,-179.297,9.053,149.571
C08521=1127.214,176.863,-62.546,-179.299,9.051,149.571
C08522=1127.219,176.614,-62.523,-179.301,9.047,149.570
C08523=1127.222,176.366,-62.499,-179.303,9.045,149.570
C08524=1127.227,176.117,-62.476,-179.306,9.042,149.570
C08525=1127.232,175.868,-62.452,-179.308,9.038,149.570
C08526=1127.236,175.619,-62.429,-179.310,9.036,149.570
C08527=1127.241,175.370,-62.406,-179.312,9.033,149.570
C08528=1127.245,175.121,-62.383,-179.314,9.029,149.570
C08529=1127.250,174.872,-62.360,-179.316,9.027,149.570
C08530=1127.255,174.624,-62.337,-179.319,9.024,149.570
C08531=1127.260,174.375,-62.313,-179.321,9.021,149.570
C08532=1127.264,174.126,-62.290,-179.323,9.017,149.569
C08533=1127.268,173.877,-62.267,-179.325,9.015,149.569
C08534=1127.273,173.628,-62.244,-179.328,9.012,149.569
C08535=1127.278,173.379,-62.220,-179.330,9.008,149.569
C08536=1127.282,173.130,-62.198,-179.332,9.006,149.569
C08537=1127.286,172.881,-62.174,-179.334,9.003,149.569
C08538=1127.291,172.632,-62.151,-179.337,9.000,149.569
C08539=1127.296,172.384,-62.128,-179.339,8.996,149.569
C08540=1127.300,172.169,-62.109,-179.341,8.994,149.569
C08541=1127.304,171.956,-62.089,-179.343,8.992,149.569
C08542=1127.308,171.740,-62.069,-179.345,8.989,149.569
C08543=1127.312,171.527,-62.049,-179.347,8.986,149.568
C08544=1127.316,171.312,-62.029,-179.349,8.984,149.568
C08545=1127.320,171.098,-62.009,-179.350,8.981,149.568
C08546=1127.324,170.884,-61.990,-179.352,8.979,149.568
C08547=1127.328,170.669,-61.969,-179.354,8.975,149.568
C08548=1127.332,170.420,-61.947,-179.357,8.972,149.568
C08549=1127.337,170.172,-61.924,-179.359,8.970,149.568
C08550=1127.342,169.923,-61.901,-179.361,8.967,149.568
C08551=1127.346,169.674,-61.878,-179.363,8.963,149.568
C08552=1127.351,169.424,-61.855,-179.366,8.960,149.568
C08553=1127.356,169.175,-61.832,-179.369,8.957,149.568
C08554=1127.360,168.927,-61.810,-179.371,8.954,149.568
C08555=1127.365,168.678,-61.786,-179.373,8.951,149.567
C08556=1127.369,168.429,-61.764,-179.375,8.948,149.567
C08557=1127.374,168.180,-61.741,-179.378,8.945,149.567
C08558=1127.378,167.931,-61.718,-179.380,8.942,149.567
C08559=1127.383,167.683,-61.695,-179.382,8.939,149.567
C08560=1127.388,167.433,-61.672,-179.385,8.935,149.567
C08561=1127.392,167.184,-61.650,-179.387,8.932,149.567
C08562=1127.397,166.936,-61.627,-179.390,8.929,149.567
C08563=1127.402,166.687,-61.605,-179.392,8.926,149.567
C08564=1127.406,166.438,-61.581,-179.394,8.923,149.567
C08565=1127.411,166.188,-61.559,-179.397,8.920,149.567
C08566=1127.416,165.940,-61.536,-179.399,8.917,149.567
C08567=1127.420,165.691,-61.513,-179.401,8.914,149.566
C08568=1127.425,165.442,-61.491,-179.403,8.911,149.566
C08569=1127.429,165.194,-61.468,-179.406,8.907,149.566
C08570=1127.435,164.944,-61.446,-179.408,8.904,149.566
C08571=1127.438,164.695,-61.423,-179.411,8.901,149.566
C08572=1127.443,164.446,-61.401,-179.413,8.898,149.566
C08573=1127.448,164.197,-61.378,-179.416,8.895,149.566
C08574=1127.452,163.948,-61.356,-179.418,8.891,149.566
C08575=1127.457,163.699,-61.333,-179.420,8.888,149.566
C08576=1127.462,163.450,-61.311,-179.423,8.885,149.566
C08577=1127.467,163.201,-61.288,-179.425,8.882,149.566
C08578=1127.471,162.952,-61.265,-179.428,8.878,149.565
C08579=1127.475,162.704,-61.243,-179.430,8.875,149.565
C08580=1127.480,162.454,-61.220,-179.433,8.871,149.565
C08581=1127.484,162.206,-61.198,-179.435,8.868,149.565
C08582=1127.489,161.957,-61.176,-179.438,8.865,149.565
C08583=1127.494,161.707,-61.153,-179.440,8.862,149.565
C08584=1127.499,161.459,-61.131,-179.443,8.859,149.565
C08585=1127.503,161.210,-61.109,-179.445,8.855,149.565
C08586=1127.508,160.960,-61.086,-179.447,8.852,149.565
C08587=1127.513,160.712,-61.064,-179.450,8.849,149.565
C08588=1127.517,160.463,-61.042,-179.452,8.845,149.564
C08589=1127.522,160.213,-61.019,-179.455,8.842,149.564
C08590=1127.526,159.965,-60.997,-179.458,8.838,149.564
C08591=1127.531,159.716,-60.975,-179.460,8.835,149.564
C08592=1127.536,159.467,-60.953,-179.462,8.832,149.564
C08593=1127.541,159.218,-60.930,-179.465,8.829,149.564
C08594=1127.545,158.970,-60.908,-179.467,8.824,149.564
C08595=1127.549,158.720,-60.886,-179.470,8.821,149.564
C08596=1127.554,158.506,-60.867,-179.472,8.819,149.564
C08597=1127.558,158.292,-60.848,-179.474,8.816,149.564
C08598=1127.561,158.076,-60.829,-179.476,8.812,149.564
C08599=1127.565,157.862,-60.810,-179.478,8.810,149.564
C08600=1127.570,157.648,-60.791,-179.480,8.807,149.563
C08601=1127.574,157.434,-60.772,-179.483,8.803,149.563
C08602=1127.577,157.219,-60.752,-179.485,8.801,149.563
C08603=1127.581,157.005,-60.733,-179.487,8.798,149.563
C08604=1127.586,156.756,-60.712,-179.489,8.795,149.563
C08605=1127.591,156.507,-60.689,-179.493,8.791,149.563
C08606=1127.596,156.258,-60.667,-179.495,8.787,149.563
C08607=1127.600,156.009,-60.645,-179.497,8.784,149.563
C08608=1127.605,155.760,-60.623,-179.499,8.781,149.562
C08609=1127.609,155.511,-60.601,-179.502,8.777,149.562
C08610=1127.614,155.262,-60.580,-179.505,8.774,149.562
C08611=1127.619,155.013,-60.558,-179.507,8.770,149.562
C08612=1127.623,154.764,-60.536,-179.510,8.766,149.562
C08613=1127.628,154.514,-60.513,-179.512,8.763,149.562
C08614=1127.633,154.266,-60.492,-179.515,8.759,149.562
C08615=1127.638,154.017,-60.470,-179.517,8.755,149.562
C08616=1127.642,153.768,-60.448,-179.520,8.752,149.562
C08617=1127.647,153.519,-60.426,-179.523,8.748,149.561
C08618=1127.652,153.270,-60.404,-179.525,8.745,149.561
C08619=1127.656,153.021,-60.383,-179.528,8.741,149.561
C08620=1127.661,152.772,-60.361,-179.530,8.738,149.561
C08621=1127.666,152.523,-60.339,-179.533,8.733,149.561
C08622=1127.671,152.274,-60.318,-179.536,8.730,149.561
C08623=1127.675,152.024,-60.296,-179.538,8.727,149.561
C08624=1127.680,151.776,-60.274,-179.541,8.723,149.561
C08625=1127.684,151.526,-60.252,-179.543,8.719,149.560
C08626=1127.689,151.278,-60.230,-179.546,8.715,149.560
C08627=1127.694,151.029,-60.209,-179.548,8.712,149.560
C08628=1127.698,150.779,-60.187,-179.551,8.708,149.560
C08629=1127.703,150.531,-60.166,-179.554,8.704,149.560
C08630=1127.708,150.282,-60.144,-179.557,8.701,149.560
C08631=1127.712,150.033,-60.122,-179.559,8.696,149.560
C08632=1127.718,149.783,-60.101,-179.561,8.693,149.559
C08633=1127.722,149.535,-60.079,-179.565,8.689,149.559
C08634=1127.726,149.286,-60.058,-179.567,8.686,149.559
C08635=1127.731,149.036,-60.037,-179.569,8.681,149.559
C08636=1127.736,148.788,-60.015,-179.573,8.677,149.559
C08637=1127.740,148.538,-59.993,-179.575,8.674,149.559
C08638=1127.746,148.289,-59.972,-179.578,8.670,149.558
C08639=1127.750,148.041,-59.951,-179.580,8.667,149.558
C08640=1127.755,147.791,-59.928,-179.583,8.662,149.558
C08641=1127.759,147.542,-59.908,-179.585,8.658,149.558
C08642=1127.764,147.294,-59.886,-179.588,8.655,149.558
C08643=1127.769,147.044,-59.865,-179.590,8.651,149.558
C08644=1127.773,146.795,-59.843,-179.593,8.646,149.557
C08645=1127.779,146.546,-59.822,-179.596,8.642,149.557
C08646=1127.783,146.297,-59.801,-179.598,8.639,149.557
C08647=1127.788,146.048,-59.780,-179.601,8.635,149.557
C08648=1127.792,145.799,-59.758,-179.604,8.630,149.557
C08649=1127.797,145.550,-59.737,-179.607,8.627,149.557
C08650=1127.801,145.301,-59.716,-179.609,8.623,149.556
C08651=1127.807,145.052,-59.695,-179.612,8.619,149.556
C08652=1127.811,144.838,-59.676,-179.613,8.616,149.556
C08653=1127.814,144.623,-59.658,-179.614,8.613,149.555
C08654=1127.819,144.408,-59.640,-179.616,8.610,149.555
C08655=1127.822,144.194,-59.622,-179.617,8.607,149.555
C08656=1127.827,143.979,-59.604,-179.618,8.605,149.555
C08657=1127.831,143.764,-59.586,-179.619,8.601,149.554
C08658=1127.835,143.550,-59.567,-179.621,8.599,149.554
C08659=1127.839,143.336,-59.549,-179.622,8.596,149.553
C08660=1127.843,143.087,-59.528,-179.623,8.593,149.553
C08661=1127.849,142.837,-59.507,-179.625,8.589,149.553
C08662=1127.853,142.588,-59.485,-179.626,8.586,149.553
C08663=1127.857,142.339,-59.465,-179.628,8.582,149.552
C08664=1127.862,142.090,-59.444,-179.629,8.579,149.552
C08665=1127.867,141.841,-59.422,-179.631,8.576,149.551
C08666=1127.872,141.592,-59.402,-179.632,8.573,149.551
C08667=1127.877,141.343,-59.381,-179.634,8.569,149.551
C08668=1127.880,141.094,-59.359,-179.635,8.566,149.550
C08669=1127.886,140.845,-59.339,-179.637,8.563,149.550
C08670=1127.891,140.596,-59.318,-179.638,8.560,149.550
C08671=1127.895,140.347,-59.297,-179.640,8.557,149.550
C08672=1127.900,140.098,-59.275,-179.641,8.553,149.549
C08673=1127.905,139.849,-59.255,-179.643,8.550,149.549
C08674=1127.910,139.600,-59.234,-179.644,8.546,149.548
C08675=1127.914,139.350,-59.213,-179.646,8.544,149.548
C08676=1127.918,139.101,-59.192,-179.647,8.540,149.548
C08677=1127.924,138.852,-59.171,-179.649,8.537,149.548
C08678=1127.928,138.603,-59.150,-179.650,8.533,149.547
C08679=1127.933,138.354,-59.129,-179.652,8.531,149.547
C08680=1127.938,138.105,-59.109,-179.654,8.527,149.546
C08681=1127.943,137.856,-59.088,-179.655,8.524,149.546
C08682=1127.947,137.607,-59.067,-179.657,8.520,149.546
C08683=1127.952,137.358,-59.046,-179.659,8.517,149.546
C08684=1127.956,137.109,-59.025,-179.660,8.514,149.545
C08685=1127.961,136.859,-59.004,-179.662,8.510,149.545
C08686=1127.966,136.610,-58.984,-179.663,8.507,149.544
C08687=1127.971,136.361,-58.963,-179.665,8.503,149.544
C08688=1127.975,136.112,-58.943,-179.666,8.501,149.544
C08689=1127.980,135.863,-58.922,-179.668,8.497,149.544
C08690=1127.985,135.614,-58.901,-179.669,8.494,149.543
C08691=1127.990,135.365,-58.880,-179.671,8.490,149.543
C08692=1127.994,135.116,-58.860,-179.672,8.488,149.543
C08693=1128.000,134.866,-58.839,-179.675,8.484,149.542
C08694=1128.004,134.617,-58.819,-179.676,8.481,149.542
C08695=1128.008,134.369,-58.798,-179.678,8.478,149.542
C08696=1128.014,134.119,-58.777,-179.679,8.474,149.541
C08697=1128.018,133.870,-58.757,-179.681,8.471,149.541
C08698=1128.023,133.621,-58.736,-179.683,8.467,149.541
C08699=1128.028,133.372,-58.716,-179.684,8.464,149.540
C08700=1128.032,133.123,-58.695,-179.686,8.461,149.540
C08701=1128.037,132.874,-58.674,-179.687,8.458,149.540
C08702=1128.042,132.625,-58.654,-179.689,8.454,149.540
C08703=1128.047,132.376,-58.633,-179.691,8.451,149.539
C08704=1128.051,132.127,-58.613,-179.692,8.448,149.539
C08705=1128.056,131.878,-58.592,-179.694,8.444,149.539
C08706=1128.061,131.629,-58.571,-179.696,8.441,149.539
C08707=1128.065,131.380,-58.551,-179.698,8.438,149.538
C08708=1128.069,131.164,-58.534,-179.699,8.435,149.538
C08709=1128.074,130.950,-58.515,-179.700,8.432,149.538
C08710=1128.077,130.735,-58.498,-179.701,8.429,149.537
C08711=1128.082,130.521,-58.481,-179.703,8.427,149.537
C08712=1128.086,130.306,-58.463,-179.705,8.423,149.537
C08713=1128.090,130.091,-58.445,-179.706,8.421,149.537
C08714=1128.094,129.876,-58.428,-179.708,8.418,149.537
C08715=1128.098,129.663,-58.410,-179.709,8.415,149.536
C08716=1128.103,129.414,-58.390,-179.711,8.412,149.536
C08717=1128.108,129.164,-58.370,-179.712,8.409,149.536
C08718=1128.113,128.915,-58.349,-179.714,8.405,149.535
C08719=1128.117,128.666,-58.329,-179.716,8.402,149.535
C08720=1128.122,128.417,-58.308,-179.718,8.398,149.535
C08721=1128.127,128.168,-58.288,-179.720,8.395,149.535
C08722=1128.131,127.918,-58.268,-179.721,8.392,149.534
C08723=1128.136,127.669,-58.248,-179.723,8.389,149.534
C08724=1128.141,127.420,-58.227,-179.725,8.385,149.534
C08725=1128.146,127.170,-58.207,-179.726,8.382,149.533
C08726=1128.151,126.922,-58.187,-179.728,8.379,149.533
C08727=1128.155,126.673,-58.167,-179.730,8.375,149.533
C08728=1128.160,126.423,-58.147,-179.731,8.372,149.533
C08729=1128.164,126.175,-58.127,-179.733,8.369,149.532
C08730=1128.170,125.925,-58.106,-179.735,8.365,149.532
C08731=1128.174,125.676,-58.086,-179.737,8.362,149.532
C08732=1128.179,125.427,-58.066,-179.739,8.358,149.531
C08733=1128.183,125.178,-58.045,-179.741,8.355,149.531
C08734=1128.188,124.929,-58.026,-179.743,8.351,149.531
C08735=1128.193,124.680,-58.005,-179.744,8.349,149.531
C08736=1128.198,124.430,-57.985,-179.746,8.345,149.531
C08737=1128.203,124.181,-57.965,-179.748,8.341,149.530
C08738=1128.208,123.932,-57.945,-179.749,8.339,149.530
C08739=1128.212,123.683,-57.925,-179.751,8.335,149.530
C08740=1128.216,123.434,-57.904,-179.753,8.332,149.529
C08741=1128.222,123.185,-57.885,-179.755,8.328,149.529
C08742=1128.226,122.936,-57.865,-179.756,8.325,149.529
C08743=1128.231,122.686,-57.845,-179.759,8.322,149.529
C08744=1128.235,122.437,-57.825,-179.761,8.318,149.528
C08745=1128.240,122.188,-57.805,-179.763,8.315,149.528
C08746=1128.245,121.939,-57.786,-179.764,8.312,149.528
C08747=1128.250,121.690,-57.765,-179.766,8.308,149.527
C08748=1128.255,121.440,-57.745,-179.768,8.305,149.527
C08749=1128.260,121.191,-57.725,-179.770,8.301,149.527
C08750=1128.265,120.942,-57.705,-179.771,8.298,149.527
C08751=1128.270,120.693,-57.685,-179.773,8.295,149.527
C08752=1128.274,120.444,-57.666,-179.775,8.291,149.526
C08753=1128.279,120.194,-57.646,-179.777,8.287,149.526
C08754=1128.284,119.945,-57.625,-179.779,8.284,149.526
C08755=1128.289,119.696,-57.606,-179.781,8.281,149.525
C08756=1128.294,119.447,-57.587,-179.783,8.278,149.525
C08757=1128.298,119.198,-57.566,-179.784,8.274,149.525
C08758=1128.303,118.948,-57.547,-179.786,8.270,149.525
C08759=1128.307,118.700,-57.528,-179.788,8.267,149.524
C08760=1128.312,118.451,-57.507,-179.790,8.263,149.524
C08761=1128.317,118.201,-57.488,-179.792,8.261,149.524
C08762=1128.322,117.952,-57.468,-179.793,8.257,149.524
C08763=1128.326,117.703,-57.448,-179.796,8.253,149.523
C08764=1128.330,117.488,-57.431,-179.797,8.251,149.523
C08765=1128.335,117.274,-57.414,-179.799,8.247,149.523
C08766=1128.339,117.059,-57.397,-179.800,8.244,149.523
C08767=1128.343,116.844,-57.380,-179.802,8.242,149.522
C08768=1128.347,116.629,-57.364,-179.804,8.238,149.522
C08769=1128.351,116.414,-57.346,-179.805,8.235,149.522
C08770=1128.356,116.200,-57.330,-179.807,8.233,149.522
C08771=1128.360,115.985,-57.313,-179.809,8.229,149.522
C08772=1128.365,115.736,-57.293,-179.811,8.226,149.521
C08773=1128.369,115.487,-57.274,-179.813,8.222,149.521
C08774=1128.374,115.237,-57.254,-179.814,8.219,149.521
C08775=1128.379,114.989,-57.235,-179.816,8.216,149.520
C08776=1128.384,114.739,-57.215,-179.818,8.212,149.520
C08777=1128.388,114.489,-57.195,-179.820,8.209,149.520
C08778=1128.394,114.241,-57.176,-179.822,8.205,149.520
C08779=1128.398,113.991,-57.157,-179.824,8.201,149.519
C08780=1128.402,113.742,-57.137,-179.826,8.198,149.519
C08781=1128.408,113.494,-57.117,-179.828,8.194,149.519
C08782=1128.412,113.244,-57.098,-179.830,8.191,149.519
C08783=1128.418,112.995,-57.078,-179.832,8.187,149.518
C08784=1128.422,112.746,-57.059,-179.834,8.183,149.518
C08785=1128.426,112.496,-57.040,-179.836,8.180,149.518
C08786=1128.432,112.247,-57.020,-179.838,8.176,149.518
C08787=1128.437,111.998,-57.001,-179.840,8.173,149.517
C08788=1128.441,111.749,-56.982,-179.842,8.169,149.517
C08789=1128.446,111.500,-56.962,-179.844,8.165,149.517
C08790=1128.451,111.250,-56.943,-179.846,8.162,149.517
C08791=1128.456,111.001,-56.923,-179.848,8.158,149.516
C08792=1128.460,110.752,-56.904,-179.850,8.155,149.516
C08793=1128.465,110.503,-56.885,-179.852,8.151,149.516
C08794=1128.470,110.253,-56.866,-179.855,8.147,149.516
C08795=1128.475,110.004,-56.847,-179.857,8.143,149.515
C08796=1128.480,109.755,-56.828,-179.860,8.140,149.515
C08797=1128.485,109.506,-56.809,-179.862,8.135,149.515
C08798=1128.489,109.257,-56.789,-179.865,8.131,149.515
C08799=1128.494,109.008,-56.770,-179.867,8.128,149.515
C08800=1128.499,108.758,-56.751,-179.870,8.123,149.515
C08801=1128.504,108.509,-56.733,-179.872,8.120,149.514
C08802=1128.509,108.260,-56.713,-179.875,8.116,149.514
C08803=1128.513,108.010,-56.694,-179.877,8.111,149.514
C08804=1128.518,107.761,-56.675,-179.879,8.108,149.514
C08805=1128.523,107.513,-56.655,-179.882,8.104,149.513
C08806=1128.528,107.263,-56.637,-179.884,8.100,149.513
C08807=1128.533,107.014,-56.618,-179.887,8.096,149.513
C08808=1128.537,106.765,-56.599,-179.889,8.092,149.513
C08809=1128.543,106.515,-56.580,-179.892,8.088,149.513
C08810=1128.547,106.266,-56.561,-179.894,8.083,149.512
C08811=1128.552,106.017,-56.542,-179.896,8.080,149.512
C08812=1128.556,105.768,-56.523,-179.899,8.076,149.512
C08813=1128.562,105.518,-56.504,-179.901,8.072,149.511
C08814=1128.566,105.269,-56.485,-179.903,8.068,149.511
C08815=1128.571,105.019,-56.466,-179.905,8.064,149.511
C08816=1128.576,104.771,-56.448,-179.908,8.060,149.511
C08817=1128.581,104.521,-56.428,-179.910,8.056,149.510
C08818=1128.586,104.272,-56.410,-179.912,8.053,149.510
C08819=1128.590,104.023,-56.390,-179.914,8.048,149.510
C08820=1128.595,103.808,-56.375,-179.916,8.044,149.510
C08821=1128.599,103.593,-56.358,-179.918,8.041,149.509
C08822=1128.603,103.378,-56.343,-179.919,8.038,149.509
C08823=1128.607,103.164,-56.326,-179.922,8.035,149.509
C08824=1128.611,102.949,-56.310,-179.924,8.031,149.509
C08825=1128.615,102.734,-56.293,-179.925,8.027,149.508
C08826=1128.619,102.519,-56.278,-179.927,8.024,149.508
C08827=1128.624,102.304,-56.262,-179.929,8.020,149.508
C08828=1128.628,102.055,-56.243,-179.931,8.017,149.508
C08829=1128.634,101.805,-56.224,-179.933,8.013,149.507
C08830=1128.639,101.557,-56.206,-179.936,8.009,149.507
C08831=1128.643,101.307,-56.187,-179.937,8.005,149.507
C08832=1128.648,101.058,-56.168,-179.939,8.001,149.506
C08833=1128.653,100.809,-56.150,-179.942,7.997,149.506
C08834=1128.657,100.559,-56.132,-179.944,7.993,149.506
C08835=1128.663,100.310,-56.112,-179.945,7.989,149.505
C08836=1128.668,100.061,-56.094,-179.947,7.985,149.505
C08837=1128.672,99.811,-56.076,-179.949,7.981,149.505
C08838=1128.677,99.562,-56.057,-179.951,7.977,149.504
C08839=1128.682,99.313,-56.039,-179.954,7.973,149.504
C08840=1128.687,99.064,-56.021,-179.955,7.969,149.503
C08841=1128.691,98.814,-56.002,-179.957,7.965,149.503
C08842=1128.697,98.565,-55.983,-179.960,7.961,149.503
C08843=1128.702,98.316,-55.965,-179.961,7.957,149.502
C08844=1128.706,98.067,-55.946,-179.963,7.953,149.502
C08845=1128.711,97.817,-55.928,-179.965,7.950,149.502
C08846=1128.716,97.568,-55.910,-179.967,7.945,149.501
C08847=1128.721,97.319,-55.892,-179.969,7.941,149.501
C08848=1128.726,97.069,-55.873,-179.971,7.937,149.501
C08849=1128.730,96.820,-55.855,-179.972,7.934,149.500
C08850=1128.736,96.571,-55.836,-179.975,7.929,149.500
C08851=1128.741,96.322,-55.818,-179.976,7.925,149.499
C08852=1128.746,96.072,-55.800,-179.978,7.921,149.499
C08853=1128.750,95.823,-55.782,-179.980,7.918,149.499
C08854=1128.755,95.573,-55.764,-179.981,7.914,149.498
C08855=1128.759,95.325,-55.745,-179.984,7.909,149.498
C08856=1128.765,95.075,-55.726,-179.985,7.905,149.498
C08857=1128.770,94.826,-55.709,-179.987,7.901,149.497
C08858=1128.774,94.576,-55.690,-179.989,7.897,149.497
C08859=1128.779,94.327,-55.672,-179.990,7.893,149.496
C08860=1128.784,94.078,-55.654,-179.992,7.890,149.496
C08861=1128.789,93.829,-55.636,-179.994,7.886,149.496
C08862=1128.794,93.580,-55.618,-179.996,7.881,149.495
C08863=1128.799,93.330,-55.600,-179.998,7.878,149.495
C08864=1128.803,93.080,-55.582,-179.999,7.874,149.494
C08865=1128.808,92.831,-55.564,179.999,7.870,149.494
C08866=1128.814,92.582,-55.545,179.998,7.866,149.493
C08867=1128.819,92.333,-55.527,179.996,7.862,149.493
C08868=1128.824,92.083,-55.509,179.994,7.858,149.493
C08869=1128.829,91.834,-55.491,179.993,7.854,149.492
C08870=1128.833,91.585,-55.473,179.991,7.850,149.492
C08871=1128.838,91.336,-55.455,179.990,7.846,149.491
C08872=1128.843,91.086,-55.437,179.988,7.843,149.491
C08873=1128.848,90.837,-55.419,179.986,7.839,149.490
C08874=1128.852,90.588,-55.401,179.985,7.834,149.490
C08875=1128.857,90.339,-55.383,179.984,7.830,149.489
C08876=1128.862,90.123,-55.369,179.982,7.828,149.489
C08877=1128.866,89.908,-55.353,179.981,7.824,149.489
C08878=1128.870,89.694,-55.338,179.980,7.821,149.488
C08879=1128.874,89.479,-55.322,179.978,7.817,149.488
C08880=1128.878,89.264,-55.307,179.977,7.814,149.487
C08881=1128.883,89.049,-55.291,179.976,7.810,149.487
C08882=1128.887,88.834,-55.275,179.974,7.807,149.487
C08883=1128.891,88.618,-55.261,179.973,7.804,149.486
C08884=1128.896,88.369,-55.243,179.972,7.800,149.486
C08885=1128.901,88.120,-55.225,179.970,7.796,149.485
C08886=1128.906,87.871,-55.207,179.969,7.792,149.485
C08887=1128.911,87.622,-55.189,179.967,7.788,149.484
C08888=1128.915,87.372,-55.172,179.966,7.784,149.484
C08889=1128.920,87.123,-55.154,179.964,7.780,149.483
C08890=1128.925,86.874,-55.136,179.964,7.777,149.483
C08891=1128.930,86.625,-55.118,179.962,7.773,149.483
C08892=1128.935,86.375,-55.101,179.960,7.769,149.482
C08893=1128.940,86.126,-55.083,179.959,7.765,149.481
C08894=1128.945,85.877,-55.065,179.958,7.761,149.481
C08895=1128.950,85.627,-55.048,179.956,7.757,149.481
C08896=1128.954,85.378,-55.030,179.956,7.753,149.480
C08897=1128.959,85.129,-55.012,179.954,7.749,149.480
C08898=1128.965,84.879,-54.995,179.952,7.746,149.479
C08899=1128.969,84.630,-54.977,179.951,7.741,149.479
C08900=1128.974,84.381,-54.959,179.950,7.738,149.478
C08901=1128.980,84.131,-54.942,179.949,7.734,149.478
C08902=1128.984,83.882,-54.924,179.948,7.730,149.477
C08903=1128.989,83.632,-54.907,179.946,7.726,149.477
C08904=1128.994,83.383,-54.889,179.945,7.723,149.476
C08905=1128.999,83.134,-54.871,179.944,7.719,149.476
C08906=1129.003,82.884,-54.854,179.942,7.715,149.475
C08907=1129.008,82.635,-54.836,179.942,7.711,149.474
C08908=1129.013,82.385,-54.819,179.940,7.707,149.474
C08909=1129.018,82.136,-54.801,179.939,7.703,149.473
C08910=1129.023,81.887,-54.785,179.938,7.700,149.473
C08911=1129.028,81.638,-54.767,179.936,7.696,149.473
C08912=1129.033,81.388,-54.749,179.935,7.692,149.472
C08913=1129.038,81.139,-54.732,179.934,7.689,149.471
C08914=1129.043,80.890,-54.715,179.933,7.684,149.471
C08915=1129.048,80.641,-54.697,179.932,7.681,149.470
C08916=1129.053,80.391,-54.680,179.931,7.677,149.470
C08917=1129.058,80.142,-54.662,179.930,7.674,149.469
C08918=1129.062,79.892,-54.645,179.929,7.670,149.469
C08919=1129.067,79.643,-54.627,179.927,7.666,149.468
C08920=1129.073,79.393,-54.610,179.927,7.662,149.468
C08921=1129.077,79.144,-54.592,179.925,7.658,149.467
C08922=1129.082,78.895,-54.575,179.925,7.655,149.467
C08923=1129.088,78.645,-54.558,179.923,7.651,149.466
C08924=1129.092,78.397,-54.541,179.923,7.647,149.465
C08925=1129.097,78.147,-54.524,179.922,7.643,149.465
C08926=1129.102,77.898,-54.506,179.921,7.640,149.464
C08927=1129.107,77.648,-54.489,179.920,7.637,149.464
C08928=1129.112,77.398,-54.472,179.919,7.633,149.463
C08929=1129.116,77.149,-54.454,179.918,7.629,149.463
C08930=1129.122,76.900,-54.437,179.917,7.625,149.462
C08931=1129.127,76.651,-54.420,179.916,7.622,149.462
C08932=1129.131,76.436,-54.405,179.914,7.618,149.461
C08933=1129.135,76.221,-54.391,179.913,7.615,149.461
C08934=1129.139,76.005,-54.376,179.913,7.612,149.460
C08935=1129.143,75.791,-54.361,179.911,7.608,149.460
C08936=1129.148,75.575,-54.346,179.910,7.605,149.459
C08937=1129.152,75.360,-54.331,179.908,7.601,149.459
C08938=1129.156,75.145,-54.316,179.907,7.598,149.459
C08939=1129.160,74.930,-54.302,179.905,7.594,149.458
C08940=1129.165,74.680,-54.285,179.904,7.590,149.458
C08941=1129.170,74.432,-54.268,179.903,7.586,149.457
C08942=1129.175,74.182,-54.250,179.901,7.582,149.457
C08943=1129.180,73.933,-54.234,179.900,7.578,149.456
C08944=1129.185,73.683,-54.216,179.898,7.574,149.456
C08945=1129.190,73.433,-54.199,179.897,7.570,149.455
C08946=1129.195,73.185,-54.182,179.896,7.567,149.455
C08947=1129.200,72.935,-54.165,179.894,7.563,149.455
C08948=1129.205,72.686,-54.148,179.893,7.559,149.454
C08949=1129.209,72.436,-54.132,179.892,7.555,149.454
C08950=1129.215,72.187,-54.115,179.890,7.551,149.453
C08951=1129.219,71.938,-54.098,179.888,7.547,149.453
C08952=1129.225,71.688,-54.081,179.887,7.543,149.452
C08953=1129.229,71.439,-54.063,179.886,7.539,149.452
C08954=1129.235,71.190,-54.046,179.884,7.535,149.451
C08955=1129.239,70.941,-54.030,179.883,7.531,149.451
C08956=1129.244,70.691,-54.012,179.881,7.527,149.450
C08957=1129.249,70.442,-53.996,179.880,7.523,149.450
C08958=1129.254,70.193,-53.980,179.878,7.519,149.449
C08959=1129.259,69.943,-53.962,179.877,7.515,149.449
C08960=1129.264,69.693,-53.946,179.876,7.511,149.448
C08961=1129.269,69.444,-53.929,179.874,7.507,149.448
C08962=1129.274,69.195,-53.912,179.873,7.503,149.447
C08963=1129.278,68.945,-53.895,179.871,7.499,149.447
C08964=1129.284,68.696,-53.878,179.870,7.495,149.446
C08965=1129.289,68.447,-53.862,179.868,7.491,149.446
C08966=1129.294,68.197,-53.845,179.867,7.487,149.445
C08967=1129.299,67.948,-53.828,179.866,7.482,149.445
C08968=1129.304,67.699,-53.812,179.864,7.479,149.444
C08969=1129.308,67.449,-53.795,179.862,7.475,149.444
C08970=1129.314,67.200,-53.778,179.861,7.471,149.443
C08971=1129.319,66.950,-53.762,179.860,7.466,149.443
C08972=1129.323,66.700,-53.745,179.858,7.463,149.442
C08973=1129.329,66.451,-53.728,179.857,7.459,149.442
C08974=1129.333,66.202,-53.712,179.855,7.454,149.441
C08975=1129.338,65.952,-53.695,179.854,7.450,149.441
C08976=1129.344,65.703,-53.678,179.852,7.447,149.440
C08977=1129.348,65.454,-53.662,179.851,7.442,149.440
C08978=1129.353,65.205,-53.645,179.850,7.438,149.439
C08979=1129.358,64.955,-53.629,179.848,7.434,149.439
C08980=1129.363,64.705,-53.612,179.847,7.431,149.439
C08981=1129.368,64.456,-53.596,179.845,7.426,149.438
C08982=1129.373,64.207,-53.579,179.844,7.422,149.438
C08983=1129.378,63.958,-53.563,179.842,7.418,149.437
C08984=1129.383,63.708,-53.547,179.841,7.414,149.436
C08985=1129.388,63.458,-53.530,179.840,7.410,149.436
C08986=1129.393,63.209,-53.513,179.838,7.406,149.436
C08987=1129.398,62.959,-53.497,179.837,7.402,149.435
C08988=1129.402,62.744,-53.483,179.836,7.399,149.435
C08989=1129.406,62.530,-53.469,179.835,7.396,149.434
C08990=1129.411,62.314,-53.454,179.833,7.392,149.434
C08991=1129.415,62.099,-53.440,179.833,7.389,149.433
C08992=1129.419,61.884,-53.425,179.831,7.385,149.433
C08993=1129.424,61.669,-53.412,179.830,7.382,149.432
C08994=1129.427,61.454,-53.398,179.828,7.378,149.432
C08995=1129.432,61.239,-53.384,179.828,7.375,149.432
C08996=1129.437,60.990,-53.367,179.826,7.371,149.431
C08997=1129.442,60.740,-53.351,179.825,7.366,149.430
C08998=1129.447,60.491,-53.335,179.823,7.363,149.430
C08999=1129.452,60.241,-53.319,179.822,7.359,149.430
C09000=1129.457,59.992,-53.302,179.821,7.354,149.429
C09001=1129.462,59.742,-53.286,179.819,7.350,149.429
C09002=1129.467,59.493,-53.270,179.818,7.347,149.428
C09003=1129.472,59.243,-53.253,179.816,7.342,149.427
C09004=1129.477,58.994,-53.238,179.815,7.338,149.427
C09005=1129.482,58.744,-53.221,179.813,7.334,149.427
C09006=1129.487,58.495,-53.206,179.812,7.330,149.426
C09007=1129.491,58.246,-53.189,179.811,7.326,149.426
C09008=1129.497,57.996,-53.173,179.810,7.322,149.425
C09009=1129.501,57.747,-53.157,179.808,7.318,149.424
C09010=1129.507,57.497,-53.141,179.806,7.314,149.424
C09011=1129.511,57.248,-53.124,179.805,7.310,149.423
C09012=1129.517,56.998,-53.109,179.804,7.306,149.423
C09013=1129.522,56.750,-53.092,179.803,7.302,149.422
C09014=1129.526,56.499,-53.077,179.801,7.298,149.422
C09015=1129.531,56.251,-53.060,179.800,7.294,149.422
C09016=1129.536,56.001,-53.044,179.798,7.289,149.421
C09017=1129.542,55.751,-53.029,179.797,7.286,149.420
C09018=1129.546,55.502,-53.012,179.796,7.281,149.420
C09019=1129.552,55.252,-52.996,179.794,7.277,149.419
C09020=1129.557,55.004,-52.980,179.793,7.273,149.419
C09021=1129.561,54.753,-52.964,179.792,7.269,149.418
C09022=1129.567,54.504,-52.949,179.790,7.265,149.418
C09023=1129.571,54.255,-52.932,179.789,7.261,149.417
C09024=1129.577,54.005,-52.916,179.787,7.257,149.417
C09025=1129.582,53.756,-52.901,179.786,7.253,149.416
C09026=1129.587,53.506,-52.884,179.785,7.249,149.416
C09027=1129.592,53.257,-52.868,179.784,7.244,149.415
C09028=1129.597,53.008,-52.854,179.782,7.241,149.415
C09029=1129.601,52.758,-52.837,179.781,7.236,149.414
C09030=1129.606,52.509,-52.821,179.779,7.232,149.414
C09031=1129.612,52.259,-52.806,179.778,7.228,149.413
C09032=1129.617,52.009,-52.790,179.777,7.224,149.413
C09033=1129.622,51.761,-52.773,179.775,7.220,149.412
C09034=1129.627,51.511,-52.758,179.774,7.216,149.411
C09035=1129.632,51.261,-52.742,179.773,7.212,149.411
C09036=1129.636,51.012,-52.727,179.771,7.208,149.410
C09037=1129.642,50.763,-52.711,179.770,7.204,149.410
C09038=1129.646,50.513,-52.695,179.769,7.199,149.409
C09039=1129.652,50.264,-52.679,179.767,7.196,149.409
C09040=1129.657,50.014,-52.663,179.766,7.191,149.408
C09041=1129.661,49.764,-52.648,179.765,7.187,149.408
C09042=1129.667,49.515,-52.632,179.764,7.183,149.407
C09043=1129.672,49.266,-52.617,179.762,7.179,149.407
C09044=1129.676,49.051,-52.603,179.762,7.176,149.406
C09045=1129.680,48.836,-52.590,179.760,7.172,149.406
C09046=1129.684,48.620,-52.576,179.759,7.169,149.405
C09047=1129.690,48.405,-52.563,179.757,7.165,149.405
C09048=1129.693,48.190,-52.549,179.757,7.162,149.404
C09049=1129.697,47.974,-52.535,179.755,7.157,149.404
C09050=1129.702,47.759,-52.522,179.755,7.154,149.403
C09051=1129.706,47.543,-52.509,179.753,7.150,149.403
C09052=1129.711,47.294,-52.494,179.752,7.146,149.402
C09053=1129.717,47.045,-52.478,179.750,7.142,149.402
C09054=1129.721,46.796,-52.463,179.749,7.138,149.401
C09055=1129.726,46.545,-52.447,179.748,7.134,149.401
C09056=1129.731,46.296,-52.431,179.747,7.129,149.400
C09057=1129.736,46.047,-52.416,179.745,7.126,149.400
C09058=1129.742,45.798,-52.401,179.744,7.121,149.399
C09059=1129.746,45.547,-52.385,179.743,7.117,149.398
C09060=1129.751,45.298,-52.370,179.741,7.113,149.398
C09061=1129.756,45.049,-52.354,179.740,7.109,149.397
C09062=1129.762,44.800,-52.339,179.739,7.105,149.397
C09063=1129.766,44.550,-52.324,179.738,7.100,149.396
C09064=1129.771,44.300,-52.308,179.737,7.096,149.396
C09065=1129.776,44.051,-52.293,179.735,7.092,149.395
C09066=1129.781,43.802,-52.277,179.734,7.088,149.395
C09067=1129.787,43.552,-52.262,179.732,7.084,149.394
C09068=1129.791,43.303,-52.247,179.731,7.080,149.393
C09069=1129.797,43.053,-52.232,179.730,7.075,149.393
C09070=1129.801,42.804,-52.216,179.729,7.071,149.392
C09071=1129.806,42.554,-52.201,179.728,7.067,149.392
C09072=1129.812,42.305,-52.185,179.727,7.063,149.391
C09073=1129.816,42.056,-52.170,179.725,7.059,149.391
C09074=1129.822,41.806,-52.155,179.724,7.055,149.390
C09075=1129.827,41.557,-52.140,179.723,7.050,149.389
C09076=1129.832,41.307,-52.125,179.721,7.046,149.389
C09077=1129.836,41.057,-52.109,179.720,7.042,149.388
C09078=1129.842,40.808,-52.094,179.719,7.037,149.388
C09079=1129.847,40.558,-52.080,179.717,7.033,149.387
C09080=1129.852,40.309,-52.064,179.716,7.029,149.387
C09081=1129.857,40.060,-52.049,179.715,7.024,149.386
C09082=1129.862,39.810,-52.033,179.713,7.021,149.386
C09083=1129.867,39.561,-52.019,179.712,7.016,149.385
C09084=1129.872,39.311,-52.003,179.711,7.012,149.384
C09085=1129.877,39.062,-51.988,179.710,7.008,149.384
C09086=1129.883,38.812,-51.974,179.709,7.004,149.383
C09087=1129.887,38.562,-51.958,179.708,6.999,149.383
C09088=1129.892,38.313,-51.943,179.706,6.995,149.382
C09089=1129.897,38.063,-51.928,179.705,6.991,149.381
C09090=1129.902,37.814,-51.913,179.704,6.987,149.381
C09091=1129.907,37.565,-51.898,179.703,6.983,149.380
C09092=1129.912,37.315,-51.884,179.702,6.978,149.380
C09093=1129.917,37.066,-51.868,179.700,6.974,149.379
C09094=1129.922,36.816,-51.854,179.699,6.970,149.378
C09095=1129.928,36.566,-51.838,179.697,6.965,149.378
C09096=1129.933,36.317,-51.824,179.696,6.961,149.377
C09097=1129.937,36.068,-51.809,179.695,6.957,149.377
C09098=1129.943,35.818,-51.793,179.694,6.952,149.376
C09099=1129.948,35.569,-51.779,179.693,6.948,149.375
C09100=1129.952,35.347,-51.766,179.692,6.944,149.375
C09101=1129.957,35.125,-51.752,179.691,6.941,149.374
C09102=1129.961,34.903,-51.739,179.690,6.936,149.374
C09103=1129.966,34.682,-51.726,179.689,6.933,149.373
C09104=1129.970,34.460,-51.713,179.688,6.929,149.373
C09105=1129.975,34.238,-51.700,179.686,6.925,149.372
C09106=1129.979,34.016,-51.687,179.686,6.921,149.372
C09107=1129.984,33.794,-51.673,179.684,6.917,149.371
C09108=1129.989,33.545,-51.658,179.683,6.913,149.371
C09109=1129.994,33.295,-51.644,179.682,6.909,149.370
C09110=1129.999,33.045,-51.629,179.681,6.904,149.369
C09111=1130.004,32.796,-51.614,179.680,6.900,149.369
C09112=1130.009,32.546,-51.600,179.678,6.896,149.368
C09113=1130.014,32.298,-51.585,179.677,6.892,149.368
C09114=1130.020,32.048,-51.570,179.676,6.887,149.367
C09115=1130.025,31.798,-51.556,179.675,6.883,149.366
C09116=1130.029,31.549,-51.541,179.673,6.878,149.366
C09117=1130.034,31.300,-51.527,179.672,6.874,149.365
C09118=1130.040,31.050,-51.512,179.671,6.870,149.364
C09119=1130.045,30.800,-51.497,179.670,6.865,149.364
C09120=1130.068,29.678,-51.432,179.854,6.486,149.226
C09121=1130.073,29.428,-51.418,179.851,6.485,149.227
C09122=1130.077,29.179,-51.403,179.848,6.484,149.228
C09123=1130.082,28.929,-51.388,179.845,6.483,149.228
C09124=1130.088,28.680,-51.375,179.843,6.482,149.228
C09125=1130.093,28.431,-51.360,179.840,6.481,149.229
C09126=1130.098,28.181,-51.346,179.838,6.480,149.230
C09127=1130.103,27.931,-51.331,179.835,6.478,149.230
C09128=1130.108,27.682,-51.316,179.833,6.477,149.230
C09129=1130.114,27.412,-51.301,179.830,6.476,149.231
C09130=1130.119,27.144,-51.285,179.827,6.475,149.232
